                   "addrGen2":
                       // Выплнение команд генератора 2
                       REGION ADRES_GENERATOR 2     
                           CASE "GlobalDATA".REQ.CMD OF
                               "cmdSCUR":
                                   REGION SET_CURRENT
                                       //Установка тока генератора
                                       IF "GeneratorDATA_2".CMD_CP = FALSE THEN
                                           "GeneratorDATA_2".CP_Programm := "GlobalDATA".REQ.Value;
                                           "GeneratorDATA_2".CMD_CP := TRUE;
                                       END_IF;
                                       //Проверяем выполнение команды от генератора
                                       IF "GeneratorDATA_2".cmdDone = TRUE AND "GeneratorDATA_2".cmd_Nunmber = "FB_STATE_CURRENT_PROGRAMM" THEN
                                           "GlobalDATA".RESP.Value := "GeneratorDATA_2".CP_Programm;
                                           "GlobalDATA".RESP.Done := 1;
                                       ELSIF "GeneratorDATA_2".cmdError = TRUE THEN
                                           "GlobalDATA".RESP.Value := "GeneratorDATA_2".cmdState;
                                           "GlobalDATA".RESP.Done := 1;
                                       END_IF;
                                   END_REGION SET_CURRENT
                               "cmdSVLT":
                                   REGION SET_VOLTAGE
                                       //Устанавливаем напряжение генератора
                                       IF "GeneratorDATA_2".CMD_VP = FALSE THEN
                                           #TempReal := UINT_TO_REAL("GlobalDATA".REQ.Value);
                                           "GeneratorDATA_2".VP_Programm := #TempReal / 10.0;
                                           "GeneratorDATA_2".CMD_VP := TRUE;
                                       END_IF;
                                       //Проверяем выполнение команды от генератора
                                       IF "GeneratorDATA_2".cmdDone = TRUE AND "GeneratorDATA_2".cmd_Nunmber = "FB_STATE_VOLTAGE_PROGRAMM" THEN
                                           #TempReal := "GeneratorDATA_2".VP_Programm * 10.0;
                                           #TempUint := REAL_TO_UINT(#TempReal);
                                           "GlobalDATA".RESP.Value := #TempUint;
                                           "GlobalDATA".RESP.Done := 1;
                                       ELSIF "GeneratorDATA_2".cmdError = TRUE THEN
                                           "GlobalDATA".RESP.Value := "GeneratorDATA_2".cmdState;
                                           "GlobalDATA".RESP.Done := 1;
                                       END_IF;
                                   END_REGION SET_VOLTAGE
                               "cmdGCUR":
                                   REGION GET_CURRENT
                                       //Чтение тока генератора
                                       "GeneratorDATA_2".CMD_MON := TRUE;

                                       //Проверяем выполнение команды от генератора
                                       IF "GeneratorDATA_2".cmdDone = TRUE AND "GeneratorDATA_2".cmd_Nunmber = "FB_STATE_MONITOR" THEN
                                           "GlobalDATA".RESP.Value := "GeneratorDATA_2".CP_Monitor;
                                           "GlobalDATA".RESP.Done := 1;
                                       ELSIF "GeneratorDATA_2".cmdError = TRUE THEN
                                           "GlobalDATA".RESP.Value := "GeneratorDATA_2".cmdState;
                                           "GlobalDATA".RESP.Done := 1;
                                       END_IF;
                                   END_REGION GET_CURRENT
                               "cmdGVLT":
                                   REGION GET_VALUE
                                       //Чтение напряжения генератора
                                       "GeneratorDATA_2".CMD_MON := TRUE;

                                       //Проверяем выполнение команды от генератора
                                       IF "GeneratorDATA_2".cmdDone = TRUE AND "GeneratorDATA_2".cmd_Nunmber = "FB_STATE_MONITOR" THEN
                                           #TempReal := "GeneratorDATA_2".VP_Monitor * 10.0;
                                           #TempUint := REAL_TO_UINT(#TempReal);
                                           "GlobalDATA".RESP.Value := #TempUint;
                                           "GlobalDATA".RESP.Done := 1;
                                       ELSIF "GeneratorDATA_2".cmdError = TRUE THEN
                                           "GlobalDATA".RESP.Value := "GeneratorDATA_2".cmdState;
                                           "GlobalDATA".RESP.Done := 1;
                                       END_IF;
                                   END_REGION GET_VALUE
                               "cmdSRAY":
                                   REGION SET_XRAY
                                       //Включение X-RAY
                                       //Включение X-RAY если шторка находится в закрытом положении
                                       IF "GlobalDATA".Shutter2.setPOS1 OR "GlobalDATA".Shutter2.setPOS2 THEN
                                           IF "GlobalDATA".REQ.Value = 1 THEN
                                               "GlobalDATA".Generator2.CmdXRAY_ON := TRUE;
                                           ELSIF "GlobalDATA".REQ.Value = 0 THEN
                                               "GlobalDATA".Generator2.CmdXRAY_ON := FALSE;
                                           END_IF;

                                           //Проверяем статус генератора
                                           IF "GeneratorDATA_2".cmdDone = TRUE AND "GeneratorDATA_2".cmd_Nunmber = "FB_STATE_MONITOR" THEN
                                               IF ("GlobalDATA".REQ.Value = 1 AND "GlobalDATA".Generator2.XRAY_Status = TRUE) THEN
                                                   "GlobalDATA".RESP.Value := 1;
                                                   "GlobalDATA".RESP.Done := 1;
                                               END_IF;
                                               IF ("GlobalDATA".REQ.Value = 0 AND "GlobalDATA".Generator2.XRAY_Status = FALSE) THEN
                                                   "GlobalDATA".RESP.Value := 0;
                                                   "GlobalDATA".RESP.Done := 1;
                                               END_IF;
                                               IF "GeneratorDATA_2".cmdError = TRUE THEN
                                                   "GlobalDATA".RESP.Value := "GeneratorDATA_2".cmdState;
                                                   "GlobalDATA".RESP.Done := 1;
                                               END_IF;
                                           END_IF;
                                       ELSE
                                           "GlobalDATA".RESP.Value := "ERR_UNDEFINED_STATE";
                                           "GlobalDATA".RESP.Done := 1;
                                       END_IF;
                                   END_REGION SET_XRAY
                               "cmdGRAY":
                                   REGION GET_XRAY_STATUS
                                       //Проверяем статус генератора
                                       "GeneratorDATA_2".CMD_STAT := TRUE;
                                       IF "GeneratorDATA_2".cmdDone = TRUE AND "GeneratorDATA_2".cmd_Nunmber = "FB_STATE_HV_STATUS" THEN
                                           IF "GeneratorDATA_2".X_RAY_Status = TRUE THEN
                                               "GlobalDATA".RESP.Value := 1;
                                           ELSE
                                               "GlobalDATA".RESP.Value := 0;
                                           END_IF;
                                           "GlobalDATA".RESP.Done := 1;
                                       ELSIF "GeneratorDATA_2".cmdError = TRUE THEN
                                           "GlobalDATA".RESP.Value := "GeneratorDATA_2".cmdState;
                                           "GlobalDATA".REQ.CMD := 0;
                                       END_IF;
                                   END_REGION GET_XRAY_STATUS
                               "cmdSWAR":
                                   REGION SET_WARM
                                       //Установка режима прогрева генератора
                                       IF "GlobalDATA".Generator2.Ready = TRUE THEN
                                           "GlobalDATA".Generator2.cmdWarm := "GlobalDATA".REQ.Value;
                                           IF "GlobalDATA".Generator2.warmEN THEN
                                               "GlobalDATA".RESP.Done := 1;
                                               //Возвращаем код выполнения программы без ошибок
                                               "GlobalDATA".RESP.Value := "GlobalDATA".Generator2.cmdWarm;
                                           END_IF;
                                       ELSE
                                           //Если генератор был не готов, то выдаем ошибку
                                           "GlobalDATA".RESP.Done := 1;
                                           "GlobalDATA".RESP.Value := "ERR_UNDEFINED_STATE";
                                       END_IF;
                                   END_REGION SET_WARM
                               "cmdGWAR":
                                   REGION GET_WARM
                                       //Если генератор готов и идет прогрев, то возвращаем значение таблицы прогрева
                                       IF "GlobalDATA".Generator2.Ready = TRUE AND "GlobalDATA".Generator2.warmEN THEN
                                           //Возвращаем код выполнения программы без ошибок
                                           "GlobalDATA".RESP.Value := "GlobalDATA".Generator2.cmdWarm;
                                       ELSE
                                           //Если генератор был не готов или не выполняется прогрев, то выдаем ошибку
                                           "GlobalDATA".RESP.Value := "STATUS_NO_CALL";
                                       END_IF;
                                       "GlobalDATA".RESP.Done := 1;
                                   END_REGION GET_WARM
                               "cmdSCLR":
                                   REGION SET_CLEAR_FAULT
                                       //Сброс ошибок генератора
                                       "GeneratorDATA_2".CMD_CLR := TRUE;
                                       //Проверяем выполнение команды от генератора
                                       IF "GeneratorDATA_2".cmdDone = TRUE AND "GeneratorDATA_2".cmd_Nunmber = "FB_STATE_FAULT_CLEAR" THEN
                                           //Чтение ошибок генератора
                                           "GeneratorDATA_2".CMD_FLT := TRUE;
                                       END_IF;

                                       //Проверяем выполнение команды от генератора
                                       IF "GeneratorDATA_2".cmdDone = TRUE AND "GeneratorDATA_2".cmd_Nunmber = "FB_STATE_REPORT_FAULT" THEN
                                           "GlobalDATA".RESP.Value.%X0 := "GeneratorDATA_2".FLT[0];
                                           "GlobalDATA".RESP.Value.%X1 := "GeneratorDATA_2".FLT[1];
                                           "GlobalDATA".RESP.Value.%X2 := "GeneratorDATA_2".FLT[2];
                                           "GlobalDATA".RESP.Value.%X3 := "GeneratorDATA_2".FLT[3];
                                           "GlobalDATA".RESP.Value.%X4 := "GeneratorDATA_2".FLT[4];
                                           "GlobalDATA".RESP.Value.%X5 := "GeneratorDATA_2".FLT[5];
                                           "GlobalDATA".RESP.Value.%X6 := "GeneratorDATA_2".FLT[6];
                                           "GlobalDATA".RESP.Value.%X7 := "GeneratorDATA_2".FLT[7];
                                           "GlobalDATA".RESP.Value.%X8 := "GeneratorDATA_2".FLT[8];
                                           "GlobalDATA".RESP.Done := 1;
                                       ELSIF "GeneratorDATA_2".cmdError = TRUE THEN
                                           "GlobalDATA".RESP.Value := "GeneratorDATA_2".cmdState;
                                           "GlobalDATA".RESP.Done := 1;
                                       END_IF;
                                   END_REGION SET_CLEAR_FAULT
                               "cmdGFLT":
                                   REGION GET_FAULT
                                       //Чтение ошибок генератора
                                       "GeneratorDATA_2".CMD_FLT := TRUE;

                                       //Проверяем выполнение команды от генератора
                                       IF "GeneratorDATA_2".cmdDone = TRUE AND "GeneratorDATA_2".cmd_Nunmber = "FB_STATE_REPORT_FAULT" THEN
                                           "GlobalDATA".RESP.Value.%X0 := "GeneratorDATA_2".FLT[0];
                                           "GlobalDATA".RESP.Value.%X1 := "GeneratorDATA_2".FLT[1];
                                           "GlobalDATA".RESP.Value.%X2 := "GeneratorDATA_2".FLT[2];
                                           "GlobalDATA".RESP.Value.%X3 := "GeneratorDATA_2".FLT[3];
                                           "GlobalDATA".RESP.Value.%X4 := "GeneratorDATA_2".FLT[4];
                                           "GlobalDATA".RESP.Value.%X5 := "GeneratorDATA_2".FLT[5];
                                           "GlobalDATA".RESP.Value.%X6 := "GeneratorDATA_2".FLT[6];
                                           "GlobalDATA".RESP.Value.%X7 := "GeneratorDATA_2".FLT[7];
                                           "GlobalDATA".RESP.Value.%X8 := "GeneratorDATA_2".FLT[8];
                                           "GlobalDATA".RESP.Done := 1;
                                       ELSIF "GeneratorDATA_2".cmdError = TRUE THEN
                                           "GlobalDATA".RESP.Value := "GeneratorDATA_2".cmdState;
                                           "GlobalDATA".RESP.Done := 1;
                                       END_IF;
                                   END_REGION GET_FAULT
                               "cmdSRES":
                                   REGION SET_RESET
                                       //Выставляем признак сброса
                                       "GlobalDATA".cmdReset.Generator2 := TRUE;
                                       "GlobalDATA".RESP.Done := 1;
                                       "GlobalDATA".RESP.Value := "STATUS_SUBSEQUENT_CALL";
                                   END_REGION SET_RESET
                           END_CASE;
                       END_REGION ADRES_GENERATOR 2

                   "addrShutter1":
                       // Выплнение команд шторки 1
                       REGION ADRES_SHUTTER 1 
                           ;
                       END_REGION ADRES_SHUTTER 1

                   "addrShutter2":
                       // Выплнение команд шторки 2
                       REGION ADRES_SHUTTER 2    
                           ;
                       END_REGION ADRES_SHUTTER 2

                   "addrDoor":
                       // Выплнение команд двери
                       REGION ADRES_DOOR
                           CASE "GlobalDATA".REQ.CMD OF
                               "cmdSRES":
                                   REGION DriveDoorReset
                                       //Выставляем признак сброса
                                       "GlobalDATA".cmdReset.Door := TRUE;
                                       "GlobalDATA".RESP.Done := 1;
                                       "GlobalDATA".RESP.Value := "STATUS_SUBSEQUENT_CALL";
                                   END_REGION DriveDoorReset
                               ELSE  // Statement section ELSE
                                   ;
                           END_CASE;
                       END_REGION ADRES_DOOR

                   "addrDetector":
                       // Выплнение команд детекторов
                       REGION ADRES_DETECTOR    
                           CASE "GlobalDATA".REQ.CMD OF
                               "cmdSRES":
                                   REGION DetectorReset
                                       //Выставляем признак сброса
                                       "GlobalDATA".cmdReset.Detector := TRUE;
                                       "GlobalDATA".RESP.Done := 1;
                                       "GlobalDATA".RESP.Value := "STATUS_SUBSEQUENT_CALL";
                                   END_REGION DetectorReset
                               ELSE  // Statement section ELSE
                                   ;
                           END_CASE;
                       END_REGION ADRES_DETECTOR

                   "addrServoDrive1":
                       // Выполнение команд привода
                       REGION ADRES DRIVE1                      
                           CASE "GlobalDATA".REQ.CMD OF
                                   //КОманда на перемещение шторки
                               "cmdSPOS":
                                   //Даем команду на перемещение шторки
                                   IF "GlobalDATA".REQ.Value = 1 AND "TEL9_Drive1".driveStopped THEN
                                       "GlobalDATA".Shutter1.cmdPOS1 := TRUE;
                                   ELSIF "GlobalDATA".REQ.Value = 2 AND "TEL9_Drive1".driveStopped THEN
                                       "GlobalDATA".Shutter1.cmdPOS2 := TRUE;
                                   END_IF;

                                   //Проверяем положение шторки
                                   IF "GlobalDATA".REQ.Value = 1 AND "GlobalDATA".Shutter1.setPOS1 = TRUE AND "TEL9_Drive1".driveStopped = TRUE THEN
                                       "GlobalDATA".RESP.Done := 1;
                                       "GlobalDATA".RESP.Value := 1;
                                       "GlobalDATA".REQ.Value := 0;
                                   ELSIF "GlobalDATA".REQ.Value = 2 AND "GlobalDATA".Shutter1.setPOS2 = TRUE AND "TEL9_Drive1".driveStopped = TRUE THEN
                                       "GlobalDATA".RESP.Done := 1;
                                       "GlobalDATA".RESP.Value := 2;
                                       "GlobalDATA".REQ.Value := 0;
                                   END_IF;
                               "cmdSRES":
                                   REGION DriveReset
                                       //Выставляем признак сброса
                                       "GlobalDATA".cmdReset.Drive1 := TRUE;
                                       "GlobalDATA".RESP.Done := 1;
                                       "GlobalDATA".RESP.Value := "STATUS_SUBSEQUENT_CALL";
                                   END_REGION DriveReset   
                               ELSE  // Statement section ELSE
                                   ;
                           END_CASE;
                       END_REGION ADRES DRIVE1

                   "addrServoDrive2":
                       // Выполнение команд привода
                       REGION ADRES DRIVE2                      
                           CASE "GlobalDATA".REQ.CMD OF
                                   //КОманда на перемещение шторки
                               "cmdSPOS":
                                   //Даем команду на перемещение шторки
                                   IF "GlobalDATA".REQ.Value = 1 AND "TEL9_Drive2".driveStopped THEN
                                       "GlobalDATA".Shutter2.cmdPOS1 := TRUE;
                                   ELSIF "GlobalDATA".REQ.Value = 2 AND "TEL9_Drive2".driveStopped THEN
                                       "GlobalDATA".Shutter2.cmdPOS2 := TRUE;
                                   END_IF;

                                   //Проверяем положение шторки
                                   IF "GlobalDATA".REQ.Value = 1 AND "GlobalDATA".Shutter2.setPOS1 = TRUE AND "TEL9_Drive2".driveStopped = TRUE THEN
                                       "GlobalDATA".RESP.Done := 1;
                                       "GlobalDATA".RESP.Value := 1;
                                       "GlobalDATA".REQ.Value := 0;
                                   ELSIF "GlobalDATA".REQ.Value = 2 AND "GlobalDATA".Shutter2.setPOS2 = TRUE AND "TEL9_Drive2".driveStopped = TRUE THEN
                                       "GlobalDATA".RESP.Done := 1;
                                       "GlobalDATA".RESP.Value := 2;
                                       "GlobalDATA".REQ.Value := 0;
                                   END_IF;
                               "cmdSRES":
                                   REGION DriveReset
                                       //Выставляем признак сброса
                                       "GlobalDATA".cmdReset.Drive2 := TRUE;
                                       "GlobalDATA".RESP.Done := 1;
                                       "GlobalDATA".RESP.Value := "STATUS_SUBSEQUENT_CALL";
                                   END_REGION DriveReset   
                               ELSE  // Statement section ELSE
                                   ;
                           END_CASE;
                       END_REGION ADRES DRIVE2

                   ELSE  // Statement section ELSE
                       ;
               END_CASE;
           END_REGION ADDR_CMD_VALUE

   END_REGION STATE_RESPONCE
END_FUNCTION_BLOCK

FUNCTION "Val_to_Char" : Void   // FC7, SCL
{ S7_Optimized_Access := 'TRUE' }
VERSION : 0.1
   VAR_INPUT
      inValue : UInt;
   END_VAR
   VAR_OUTPUT
      charBUFF : Array[0..3] of Byte;
   END_VAR
   VAR_TEMP
      Countchar : UInt;
      StrValue : String;
      i : Int;
      tempBUFF : Array[0..3] of Byte;
      TEMP : UInt;
   END_VAR
BEGIN
   VAL_STRG(IN := #inValue,
            SIZE := 4,
            PREC := 0,
            FORMAT := 0,
            P := 1,
            OUT => #StrValue);

   #Countchar := 4;

   Strg_TO_Chars(Strg := #StrValue,
                 pChars := 0,
                 Cnt => #Countchar,
                 Chars := #tempBUFF);

   FOR #i := 0  TO 3 DO
      IF #tempBUFF[#i] = ' ' THEN // Statement section FOR
          #tempBUFF[#i] := '0';
       END_IF;
       #charBUFF[#i] := #tempBUFF[#i];
   END_FOR;
END_FUNCTION

// folder: DIO

FUNCTION "DI" : Void   // FC2, LAD
{ S7_Optimized_Access := 'TRUE' }
VERSION : 0.1
BEGIN

REGION Network 1: Чтение дискретных входов PLC и передача в глобальный блок данных
   // Первый байт дискретных входов
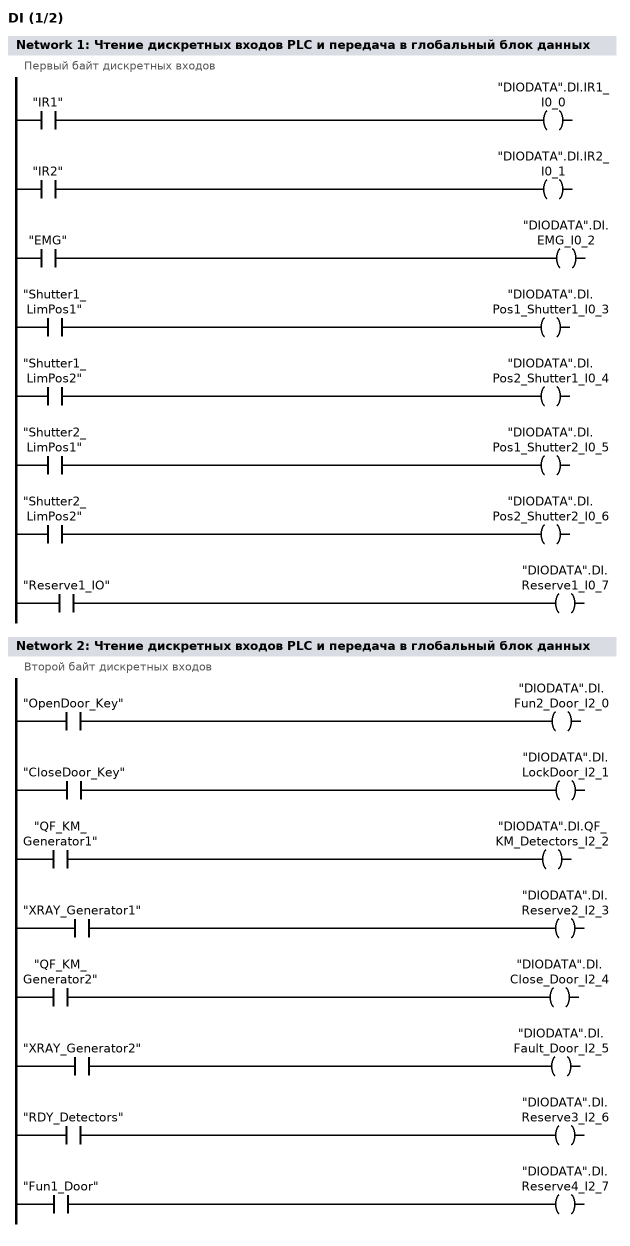
   RUNG wire#powerrail
      Contact( "IR1" )
      Coil( "DIODATA".DI.IR1_I0_0 )
   END_RUNG
   RUNG wire#powerrail
      Contact( "IR2" )
      Coil( "DIODATA".DI.IR2_I0_1 )
   END_RUNG
   RUNG wire#powerrail
      Contact( "EMG" )
      Coil( "DIODATA".DI.EMG_I0_2 )
   END_RUNG
   RUNG wire#powerrail
      Contact( "Shutter1_LimPos1" )
      Coil( "DIODATA".DI.Pos1_Shutter1_I0_3 )
   END_RUNG
   RUNG wire#powerrail
      Contact( "Shutter1_LimPos2" )
      Coil( "DIODATA".DI.Pos2_Shutter1_I0_4 )
   END_RUNG
   RUNG wire#powerrail
      Contact( "Shutter2_LimPos1" )
      Coil( "DIODATA".DI.Pos1_Shutter2_I0_5 )
   END_RUNG
   RUNG wire#powerrail
      Contact( "Shutter2_LimPos2" )
      Coil( "DIODATA".DI.Pos2_Shutter2_I0_6 )
   END_RUNG
   RUNG wire#powerrail
      Contact( "Reserve1_IO" )
      Coil( "DIODATA".DI.Reserve1_I0_7 )
   END_RUNG
   // the same network as SCL:
   "DIODATA".DI.IR1_I0_0 := "IR1";
   "DIODATA".DI.IR2_I0_1 := "IR2";
   "DIODATA".DI.EMG_I0_2 := "EMG";
   "DIODATA".DI.Pos1_Shutter1_I0_3 := "Shutter1_LimPos1";
   "DIODATA".DI.Pos2_Shutter1_I0_4 := "Shutter1_LimPos2";
   "DIODATA".DI.Pos1_Shutter2_I0_5 := "Shutter2_LimPos1";
   "DIODATA".DI.Pos2_Shutter2_I0_6 := "Shutter2_LimPos2";
   "DIODATA".DI.Reserve1_I0_7 := "Reserve1_IO";
END_REGION

REGION Network 2: Чтение дискретных входов PLC и передача в глобальный блок данных
   // Второй байт дискретных входов
   RUNG wire#powerrail
      Contact( "OpenDoor_Key" )
      Coil( "DIODATA".DI.Fun2_Door_I2_0 )
   END_RUNG
   RUNG wire#powerrail
      Contact( "CloseDoor_Key" )
      Coil( "DIODATA".DI.LockDoor_I2_1 )
   END_RUNG
   RUNG wire#powerrail
      Contact( "QF_KM_Generator1" )
      Coil( "DIODATA".DI.QF_KM_Detectors_I2_2 )
   END_RUNG
   RUNG wire#powerrail
      Contact( "XRAY_Generator1" )
      Coil( "DIODATA".DI.Reserve2_I2_3 )
   END_RUNG
   RUNG wire#powerrail
      Contact( "QF_KM_Generator2" )
      Coil( "DIODATA".DI.Close_Door_I2_4 )
   END_RUNG
   RUNG wire#powerrail
      Contact( "XRAY_Generator2" )
      Coil( "DIODATA".DI.Fault_Door_I2_5 )
   END_RUNG
   RUNG wire#powerrail
      Contact( "RDY_Detectors" )
      Coil( "DIODATA".DI.Reserve3_I2_6 )
   END_RUNG
   RUNG wire#powerrail
      Contact( "Fun1_Door" )
      Coil( "DIODATA".DI.Reserve4_I2_7 )
   END_RUNG
   // the same network as SCL:
   "DIODATA".DI.Fun2_Door_I2_0 := "OpenDoor_Key";
   "DIODATA".DI.LockDoor_I2_1 := "CloseDoor_Key";
   "DIODATA".DI.QF_KM_Detectors_I2_2 := "QF_KM_Generator1";
   "DIODATA".DI.Reserve2_I2_3 := "XRAY_Generator1";
   "DIODATA".DI.Close_Door_I2_4 := "QF_KM_Generator2";
   "DIODATA".DI.Fault_Door_I2_5 := "XRAY_Generator2";
   "DIODATA".DI.Reserve3_I2_6 := "RDY_Detectors";
   "DIODATA".DI.Reserve4_I2_7 := "Fun1_Door";
END_REGION

REGION Network 3: Чтение дискретных входов PLC и передача в глобальный блок данных
   // Третий
   //  байт дискретных входов
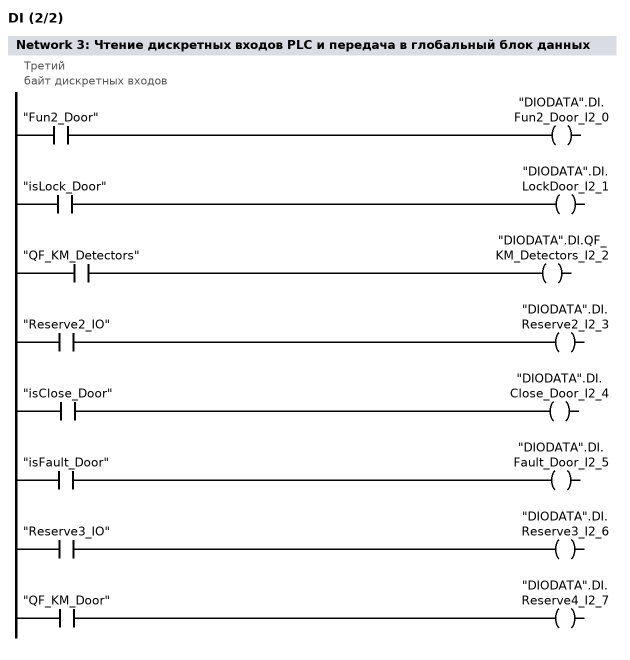
   RUNG wire#powerrail
      Contact( "Fun2_Door" )
      Coil( "DIODATA".DI.Fun2_Door_I2_0 )
   END_RUNG
   RUNG wire#powerrail
      Contact( "isLock_Door" )
      Coil( "DIODATA".DI.LockDoor_I2_1 )
   END_RUNG
   RUNG wire#powerrail
      Contact( "QF_KM_Detectors" )
      Coil( "DIODATA".DI.QF_KM_Detectors_I2_2 )
   END_RUNG
   RUNG wire#powerrail
      Contact( "Reserve2_IO" )
      Coil( "DIODATA".DI.Reserve2_I2_3 )
   END_RUNG
   RUNG wire#powerrail
      Contact( "isClose_Door" )
      Coil( "DIODATA".DI.Close_Door_I2_4 )
   END_RUNG
   RUNG wire#powerrail
      Contact( "isFault_Door" )
      Coil( "DIODATA".DI.Fault_Door_I2_5 )
   END_RUNG
   RUNG wire#powerrail
      Contact( "Reserve3_IO" )
      Coil( "DIODATA".DI.Reserve3_I2_6 )
   END_RUNG
   RUNG wire#powerrail
      Contact( "QF_KM_Door" )
      Coil( "DIODATA".DI.Reserve4_I2_7 )
   END_RUNG
   // the same network as SCL:
   "DIODATA".DI.Fun2_Door_I2_0 := "Fun2_Door";
   "DIODATA".DI.LockDoor_I2_1 := "isLock_Door";
   "DIODATA".DI.QF_KM_Detectors_I2_2 := "QF_KM_Detectors";
   "DIODATA".DI.Reserve2_I2_3 := "Reserve2_IO";
   "DIODATA".DI.Close_Door_I2_4 := "isClose_Door";
   "DIODATA".DI.Fault_Door_I2_5 := "isFault_Door";
   "DIODATA".DI.Reserve3_I2_6 := "Reserve3_IO";
   "DIODATA".DI.Reserve4_I2_7 := "QF_KM_Door";
END_REGION
END_FUNCTION

FUNCTION "DO" : Void   // FC6, LAD
{ S7_Optimized_Access := 'TRUE' }
VERSION : 0.1
BEGIN

REGION Network 1: Установка дискретных выходов PLC из глобального блока данных
   // Установка первого байта цифровых выходов
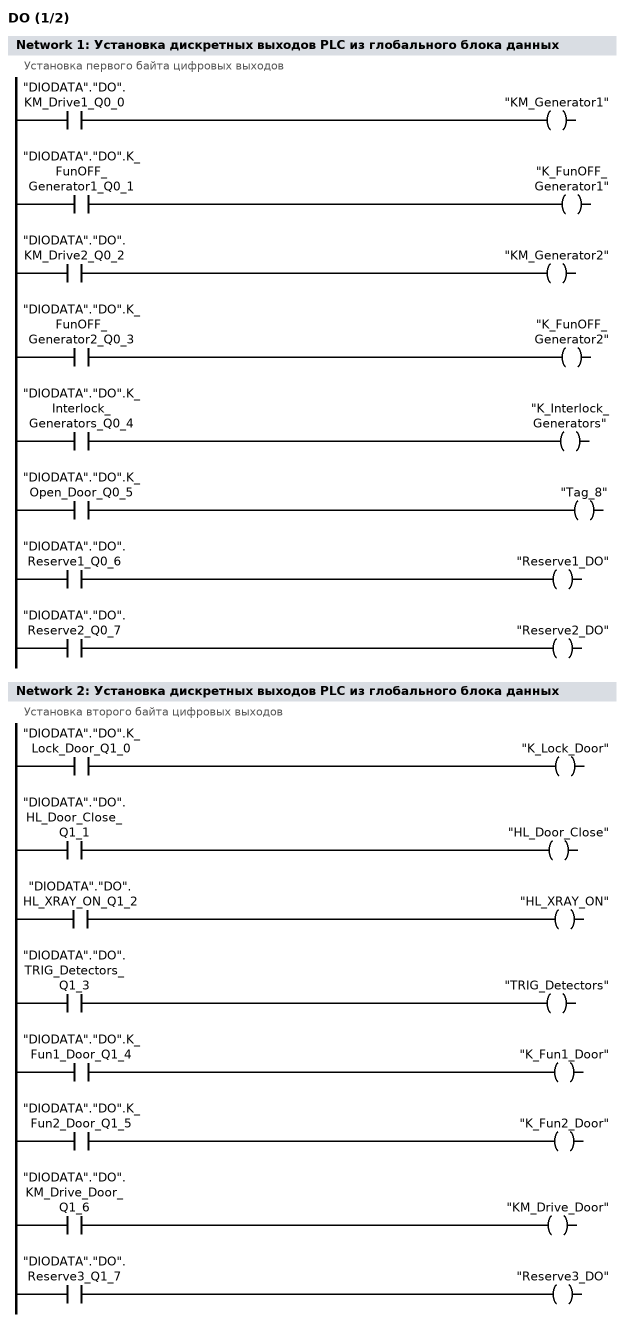
   RUNG wire#powerrail
      Contact( "DIODATA"."DO".KM_Drive1_Q0_0 )
      Coil( "KM_Generator1" )
   END_RUNG
   RUNG wire#powerrail
      Contact( "DIODATA"."DO".K_FunOFF_Generator1_Q0_1 )
      Coil( "K_FunOFF_Generator1" )
   END_RUNG
   RUNG wire#powerrail
      Contact( "DIODATA"."DO".KM_Drive2_Q0_2 )
      Coil( "KM_Generator2" )
   END_RUNG
   RUNG wire#powerrail
      Contact( "DIODATA"."DO".K_FunOFF_Generator2_Q0_3 )
      Coil( "K_FunOFF_Generator2" )
   END_RUNG
   RUNG wire#powerrail
      Contact( "DIODATA"."DO".K_Interlock_Generators_Q0_4 )
      Coil( "K_Interlock_Generators" )
   END_RUNG
   RUNG wire#powerrail
      Contact( "DIODATA"."DO".K_Open_Door_Q0_5 )
      Coil( "Tag_8" )
   END_RUNG
   RUNG wire#powerrail
      Contact( "DIODATA"."DO".Reserve1_Q0_6 )
      Coil( "Reserve1_DO" )
   END_RUNG
   RUNG wire#powerrail
      Contact( "DIODATA"."DO".Reserve2_Q0_7 )
      Coil( "Reserve2_DO" )
   END_RUNG
   // the same network as SCL:
   "KM_Generator1" := "DIODATA"."DO".KM_Drive1_Q0_0;
   "K_FunOFF_Generator1" := "DIODATA"."DO".K_FunOFF_Generator1_Q0_1;
   "KM_Generator2" := "DIODATA"."DO".KM_Drive2_Q0_2;
   "K_FunOFF_Generator2" := "DIODATA"."DO".K_FunOFF_Generator2_Q0_3;
   "K_Interlock_Generators" := "DIODATA"."DO".K_Interlock_Generators_Q0_4;
   "Tag_8" := "DIODATA"."DO".K_Open_Door_Q0_5;
   "Reserve1_DO" := "DIODATA"."DO".Reserve1_Q0_6;
   "Reserve2_DO" := "DIODATA"."DO".Reserve2_Q0_7;
END_REGION

REGION Network 2: Установка дискретных выходов PLC из глобального блока данных
   // Установка второго байта цифровых выходов
   RUNG wire#powerrail
      Contact( "DIODATA"."DO".K_Lock_Door_Q1_0 )
      Coil( "K_Lock_Door" )
   END_RUNG
   RUNG wire#powerrail
      Contact( "DIODATA"."DO".HL_Door_Close_Q1_1 )
      Coil( "HL_Door_Close" )
   END_RUNG
   RUNG wire#powerrail
      Contact( "DIODATA"."DO".HL_XRAY_ON_Q1_2 )
      Coil( "HL_XRAY_ON" )
   END_RUNG
   RUNG wire#powerrail
      Contact( "DIODATA"."DO".TRIG_Detectors_Q1_3 )
      Coil( "TRIG_Detectors" )
   END_RUNG
   RUNG wire#powerrail
      Contact( "DIODATA"."DO".K_Fun1_Door_Q1_4 )
      Coil( "K_Fun1_Door" )
   END_RUNG
   RUNG wire#powerrail
      Contact( "DIODATA"."DO".K_Fun2_Door_Q1_5 )
      Coil( "K_Fun2_Door" )
   END_RUNG
   RUNG wire#powerrail
      Contact( "DIODATA"."DO".KM_Drive_Door_Q1_6 )
      Coil( "KM_Drive_Door" )
   END_RUNG
   RUNG wire#powerrail
      Contact( "DIODATA"."DO".Reserve3_Q1_7 )
      Coil( "Reserve3_DO" )
   END_RUNG
   // the same network as SCL:
   "K_Lock_Door" := "DIODATA"."DO".K_Lock_Door_Q1_0;
   "HL_Door_Close" := "DIODATA"."DO".HL_Door_Close_Q1_1;
   "HL_XRAY_ON" := "DIODATA"."DO".HL_XRAY_ON_Q1_2;
   "TRIG_Detectors" := "DIODATA"."DO".TRIG_Detectors_Q1_3;
   "K_Fun1_Door" := "DIODATA"."DO".K_Fun1_Door_Q1_4;
   "K_Fun2_Door" := "DIODATA"."DO".K_Fun2_Door_Q1_5;
   "KM_Drive_Door" := "DIODATA"."DO".KM_Drive_Door_Q1_6;
   "Reserve3_DO" := "DIODATA"."DO".Reserve3_Q1_7;
END_REGION

REGION Network 3: Установка дискретных выходов PLC из глобального блока данных
   // Установка третьего байта цифровых выходов
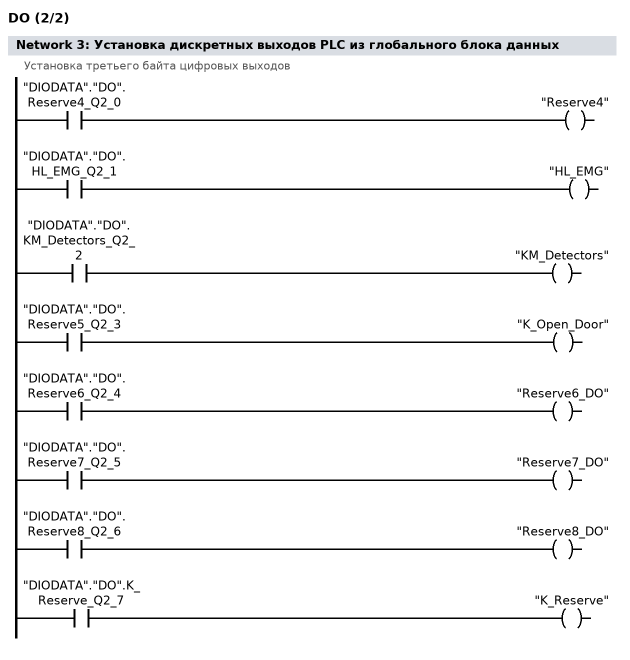
   RUNG wire#powerrail
      Contact( "DIODATA"."DO".Reserve4_Q2_0 )
      Coil( "Reserve4" )
   END_RUNG
   RUNG wire#powerrail
      Contact( "DIODATA"."DO".HL_EMG_Q2_1 )
      Coil( "HL_EMG" )
   END_RUNG
   RUNG wire#powerrail
      Contact( "DIODATA"."DO".KM_Detectors_Q2_2 )
      Coil( "KM_Detectors" )
   END_RUNG
   RUNG wire#powerrail
      Contact( "DIODATA"."DO".Reserve5_Q2_3 )
      Coil( "K_Open_Door" )
   END_RUNG
   RUNG wire#powerrail
      Contact( "DIODATA"."DO".Reserve6_Q2_4 )
      Coil( "Reserve6_DO" )
   END_RUNG
   RUNG wire#powerrail
      Contact( "DIODATA"."DO".Reserve7_Q2_5 )
      Coil( "Reserve7_DO" )
   END_RUNG
   RUNG wire#powerrail
      Contact( "DIODATA"."DO".Reserve8_Q2_6 )
      Coil( "Reserve8_DO" )
   END_RUNG
   RUNG wire#powerrail
      Contact( "DIODATA"."DO".K_Reserve_Q2_7 )
      Coil( "K_Reserve" )
   END_RUNG
   // the same network as SCL:
   "Reserve4" := "DIODATA"."DO".Reserve4_Q2_0;
   "HL_EMG" := "DIODATA"."DO".HL_EMG_Q2_1;
   "KM_Detectors" := "DIODATA"."DO".KM_Detectors_Q2_2;
   "K_Open_Door" := "DIODATA"."DO".Reserve5_Q2_3;
   "Reserve6_DO" := "DIODATA"."DO".Reserve6_Q2_4;
   "Reserve7_DO" := "DIODATA"."DO".Reserve7_Q2_5;
   "Reserve8_DO" := "DIODATA"."DO".Reserve8_Q2_6;
   "K_Reserve" := "DIODATA"."DO".K_Reserve_Q2_7;
END_REGION
END_FUNCTION

// folder: Drive

FUNCTION_BLOCK "DrivesStage"   // FB2, LAD
{ S7_Optimized_Access := 'TRUE' }
VERSION : 0.1
   VAR_INPUT
      Drive1 : Bool;   // drive 1 manage
      Drive2 : Bool;   // drive 1 manage
      Resset : Bool;   // Resset Block
      Mode : Bool;   // 0-MDI, 1-JOG
      "ON/OFF1" : Bool;   // OFF1
      JOG1 : Bool;   // JOG+
      JOG2 : Bool;   // JOG-
      cmdPOS1 : Bool;   // position to point 1
      cmdPOS2 : Bool;   // position to point 2
      Velocity : DInt;   // Velocity in MDI
      accelerationOverride : Real;   // accelerationOverride %
      decelerationOverride : Real;   // decelerationOverride %
      POS1_X : DInt;   // coordinate of point 1
      POS2_X : DInt;   // coordinate of point 2
      CmdPOS : Bool;   // CMD to traversing task
      HardWare_IO : Hw_Io;   // Hardware identifer of the drive axis
   END_VAR
   VAR_OUTPUT
      State_OFF1 : Bool;   // State OFF1
      Drive_STOP : Bool;   // State Drive Stop
      setPOS1 : Bool;   // in position 1
      setPOS2 : Bool;   // in position 2
      actualPosition : DInt;   // Current position
      Fault_Active : Bool;   // Fault Active
   END_VAR
   VAR_IN_OUT
      DATA : "typeTEL9";
   END_VAR
   VAR
      sSetPOS : Bool;
      sOFF1 : Bool;
      sOFF2 : Bool;
      sOFF3 : Bool;
      Front1 : Bool;
      Front2 : Bool;
      Front3 : Bool;
      Task : UInt;
      neg1 : Bool;
   END_VAR
   VAR_TEMP
      In_pos1 : Bool;
      In_pos2 : Bool;
   END_VAR
   VAR_TEMP   // added for the SCL form of the ladder/FBD networks
      _w1 : Bool;
      _w2 : Bool;
   END_VAR
BEGIN

REGION Network 1: Включение OFF1. Если возникает ошибка привода, то снимаем OFF1, сбрасываем ошибку и опять ввзводим OFF1
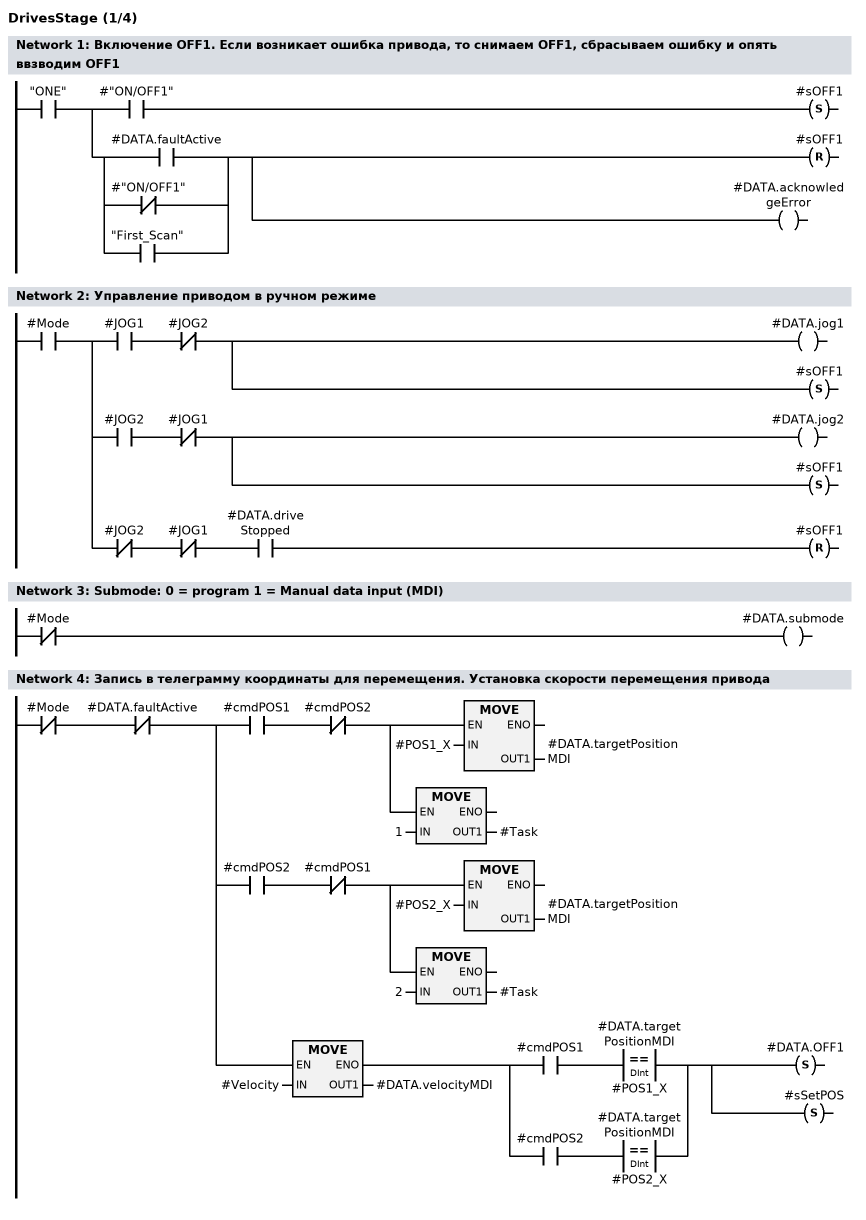
   RUNG wire#powerrail
      Contact( "ONE" )
      wire#w1
      Contact( #"ON/OFF1" )
      S_Coil( #sOFF1 )
   END_RUNG
   RUNG wire#w1
      Contact( #DATA.faultActive )
      wire#w2
      R_Coil( #sOFF1 )
   END_RUNG
   RUNG wire#w1
      I_Contact( #"ON/OFF1" )
   END_RUNG wire#w2
   RUNG wire#w1
      Contact( "First_Scan" )
   END_RUNG wire#w2
   RUNG wire#w2
      Coil( #DATA.acknowledgeError )
   END_RUNG
   // the same network as SCL:
   IF "ONE" AND #"ON/OFF1" THEN #sOFF1 := TRUE; END_IF;
   #_w1 := "ONE" AND (#DATA.faultActive OR NOT #"ON/OFF1" OR "First_Scan");
   IF #_w1 THEN #sOFF1 := FALSE; END_IF;
   #DATA.acknowledgeError := #_w1;
END_REGION

REGION Network 2: Управление приводом в ручном режиме
   RUNG wire#powerrail
      Contact( #Mode )
      wire#w1
      Contact( #JOG1 )
      I_Contact( #JOG2 )
      wire#w2
      Coil( #DATA.jog1 )
   END_RUNG
   RUNG wire#w2
      S_Coil( #sOFF1 )
   END_RUNG
   RUNG wire#w1
      Contact( #JOG2 )
      I_Contact( #JOG1 )
      wire#w3
      Coil( #DATA.jog2 )
   END_RUNG
   RUNG wire#w3
      S_Coil( #sOFF1 )
   END_RUNG
   RUNG wire#w1
      I_Contact( #JOG2 )
      I_Contact( #JOG1 )
      Contact( #DATA.driveStopped )
      R_Coil( #sOFF1 )
   END_RUNG
   // the same network as SCL:
   #DATA.jog1 := #Mode AND #JOG1 AND NOT #JOG2;
   IF #DATA.jog1 THEN #sOFF1 := TRUE; END_IF;
   #DATA.jog2 := #Mode AND #JOG2 AND NOT #JOG1;
   IF #DATA.jog2 THEN #sOFF1 := TRUE; END_IF;
   IF #Mode AND NOT #JOG2 AND NOT #JOG1 AND #DATA.driveStopped THEN #sOFF1 := FALSE; END_IF;
END_REGION

REGION Network 3: Submode: 0 = program 1 = Manual data input (MDI)
   RUNG wire#powerrail
      I_Contact( #Mode )
      Coil( #DATA.submode )
   END_RUNG
   // the same network as SCL:
   #DATA.submode := NOT #Mode;
END_REGION

REGION Network 4: Запись в телеграмму координаты для перемещения. Установка скорости перемещения привода
   RUNG wire#powerrail
      I_Contact( #Mode )
      I_Contact( #DATA.faultActive )
      wire#w1
      Contact( #cmdPOS1 )
      I_Contact( #cmdPOS2 )
      wire#w2
      Move(in := #POS1_X, out1 => #DATA.targetPositionMDI)
   END_RUNG
   RUNG wire#w2
      Move(in := 1, out1 => #Task)
   END_RUNG
   RUNG wire#w1
      Contact( #cmdPOS2 )
      I_Contact( #cmdPOS1 )
      wire#w3
      Move(in := #POS2_X, out1 => #DATA.targetPositionMDI)
   END_RUNG
   RUNG wire#w3
      Move(in := 2, out1 => #Task)
   END_RUNG
   RUNG wire#w1
      Move(in := #Velocity, out1 => #DATA.velocityMDI)
      wire#w4
      Contact( #cmdPOS1 )
      { S7_Templates := "SrcType := DInt" } EQ_Contact(in1 := #DATA.targetPositionMDI, in2 := #POS1_X)
      wire#w5
      S_Coil( #DATA.OFF1 )
   END_RUNG
   RUNG wire#w4
      Contact( #cmdPOS2 )
      { S7_Templates := "SrcType := DInt" } EQ_Contact(in1 := #DATA.targetPositionMDI, in2 := #POS2_X)
   END_RUNG wire#w5
   RUNG wire#w5
      S_Coil( #sSetPOS )
   END_RUNG
   // the same network as SCL:
   #_w1 := NOT #Mode AND NOT #DATA.faultActive;
   IF #_w1 AND #cmdPOS1 AND NOT #cmdPOS2 THEN
       #DATA.targetPositionMDI := #POS1_X;
       #Task := 1;
   END_IF;
   IF #_w1 AND #cmdPOS2 AND NOT #cmdPOS1 THEN
       #DATA.targetPositionMDI := #POS2_X;
       #Task := 2;
   END_IF;
   IF #_w1 THEN #DATA.velocityMDI := #Velocity; END_IF;
   IF #_w1 AND ((#cmdPOS1 AND (#DATA.targetPositionMDI = #POS1_X)) OR (#cmdPOS2 AND (#DATA.targetPositionMDI = #POS2_X))) THEN
       #DATA.OFF1 := TRUE;
       #sSetPOS := TRUE;
   END_IF;
END_REGION

REGION Network 5: Activate traversing task
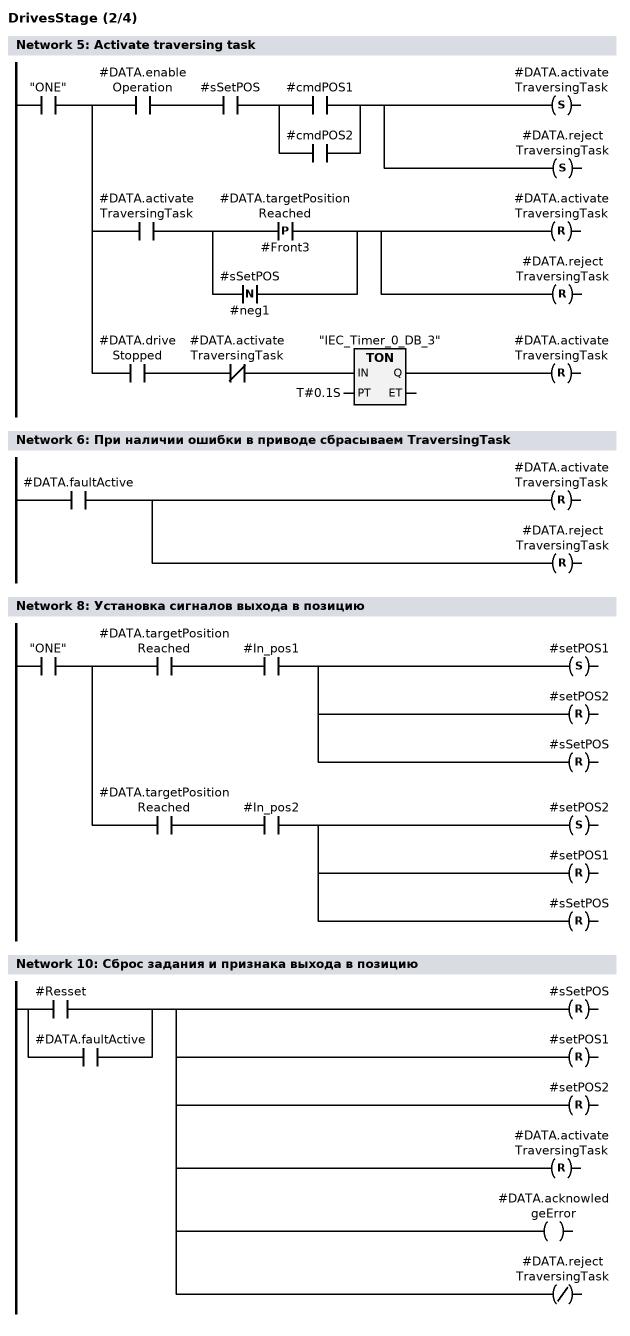
   IF "ONE" AND #DATA.enableOperation AND #sSetPOS AND (#cmdPOS1 OR #cmdPOS2) THEN
       #DATA.activateTraversingTask := TRUE;
       #DATA.rejectTraversingTask := TRUE;
   END_IF;
   #_w1 := "ONE" AND #DATA.activateTraversingTask AND #DATA.targetPositionReached AND NOT #Front3;   // rising edge of #DATA.targetPositionReached
   #Front3 := #DATA.targetPositionReached;
   #_w2 := "ONE" AND #DATA.activateTraversingTask AND NOT #sSetPOS AND #neg1;   // falling edge of #sSetPOS
   #neg1 := #sSetPOS;
   IF #_w1 OR #_w2 THEN
       #DATA.activateTraversingTask := FALSE;
       #DATA.rejectTraversingTask := FALSE;
   END_IF;
   "IEC_Timer_0_DB_3".TON(IN := "ONE" AND #DATA.driveStopped AND NOT #DATA.activateTraversingTask, PT := T#0.1S);
   IF "IEC_Timer_0_DB_3".Q THEN #DATA.activateTraversingTask := FALSE; END_IF;
END_REGION

REGION Network 6: При наличии ошибки в приводе сбрасываем TraversingTask
   RUNG wire#powerrail
      Contact( #DATA.faultActive )
      wire#w1
      R_Coil( #DATA.activateTraversingTask )
   END_RUNG
   RUNG wire#w1
      R_Coil( #DATA.rejectTraversingTask )
   END_RUNG
   // the same network as SCL:
   IF #DATA.faultActive THEN
       #DATA.activateTraversingTask := FALSE;
       #DATA.rejectTraversingTask := FALSE;
   END_IF;
END_REGION

REGION Network 7 (SCL)
   IF ABS(#DATA.actualPosition-#POS1_X)<40 THEN
       #In_pos1 := TRUE;
   ELSE
       #In_pos1 := FALSE;
   END_IF;
   IF  ABS(#DATA.actualPosition - #POS2_X) < 40 THEN
       #In_pos2 := TRUE;
   ELSE
       #In_pos2 := FALSE;
   END_IF;
END_REGION

REGION Network 8: Установка сигналов выхода в позицию
   RUNG wire#powerrail
      Contact( "ONE" )
      wire#w1
      Contact( #DATA.targetPositionReached )
      Contact( #In_pos1 )
      wire#w2
      S_Coil( #setPOS1 )
   END_RUNG
   RUNG wire#w2
      R_Coil( #setPOS2 )
   END_RUNG
   RUNG wire#w2
      R_Coil( #sSetPOS )
   END_RUNG
   RUNG wire#w1
      Contact( #DATA.targetPositionReached )
      Contact( #In_pos2 )
      wire#w3
      S_Coil( #setPOS2 )
   END_RUNG
   RUNG wire#w3
      R_Coil( #setPOS1 )
   END_RUNG
   RUNG wire#w3
      R_Coil( #sSetPOS )
   END_RUNG
   // the same network as SCL:
   IF "ONE" AND #DATA.targetPositionReached AND #In_pos1 THEN
       #setPOS1 := TRUE;
       #setPOS2 := FALSE;
       #sSetPOS := FALSE;
   END_IF;
   IF "ONE" AND #DATA.targetPositionReached AND #In_pos2 THEN
       #setPOS2 := TRUE;
       #setPOS1 := FALSE;
       #sSetPOS := FALSE;
   END_IF;
END_REGION

REGION Network 9 (SCL)
   #DATA.positioningModeMDI := 1;
   #DATA.intermediateStop := TRUE;
   #Task := 0;
END_REGION

REGION Network 10: Сброс задания и признака выхода в позицию
   RUNG wire#powerrail
      Contact( #Resset )
      wire#w1
      R_Coil( #sSetPOS )
   END_RUNG
   RUNG wire#powerrail
      Contact( #DATA.faultActive )
   END_RUNG wire#w1
   RUNG wire#w1
      R_Coil( #setPOS1 )
   END_RUNG
   RUNG wire#w1
      R_Coil( #setPOS2 )
   END_RUNG
   RUNG wire#w1
      R_Coil( #DATA.activateTraversingTask )
   END_RUNG
   RUNG wire#w1
      Coil( #DATA.acknowledgeError )
   END_RUNG
   RUNG wire#w1
      I_Coil( #DATA.rejectTraversingTask )
   END_RUNG
   // the same network as SCL:
   #_w1 := #Resset OR #DATA.faultActive;
   IF #_w1 THEN
       #sSetPOS := FALSE;
       #setPOS1 := FALSE;
       #setPOS2 := FALSE;
       #DATA.activateTraversingTask := FALSE;
   END_IF;
   #DATA.acknowledgeError := #_w1;
   #DATA.rejectTraversingTask := NOT #_w1;
END_REGION

REGION Network 11: Формирование телеграммы для привода
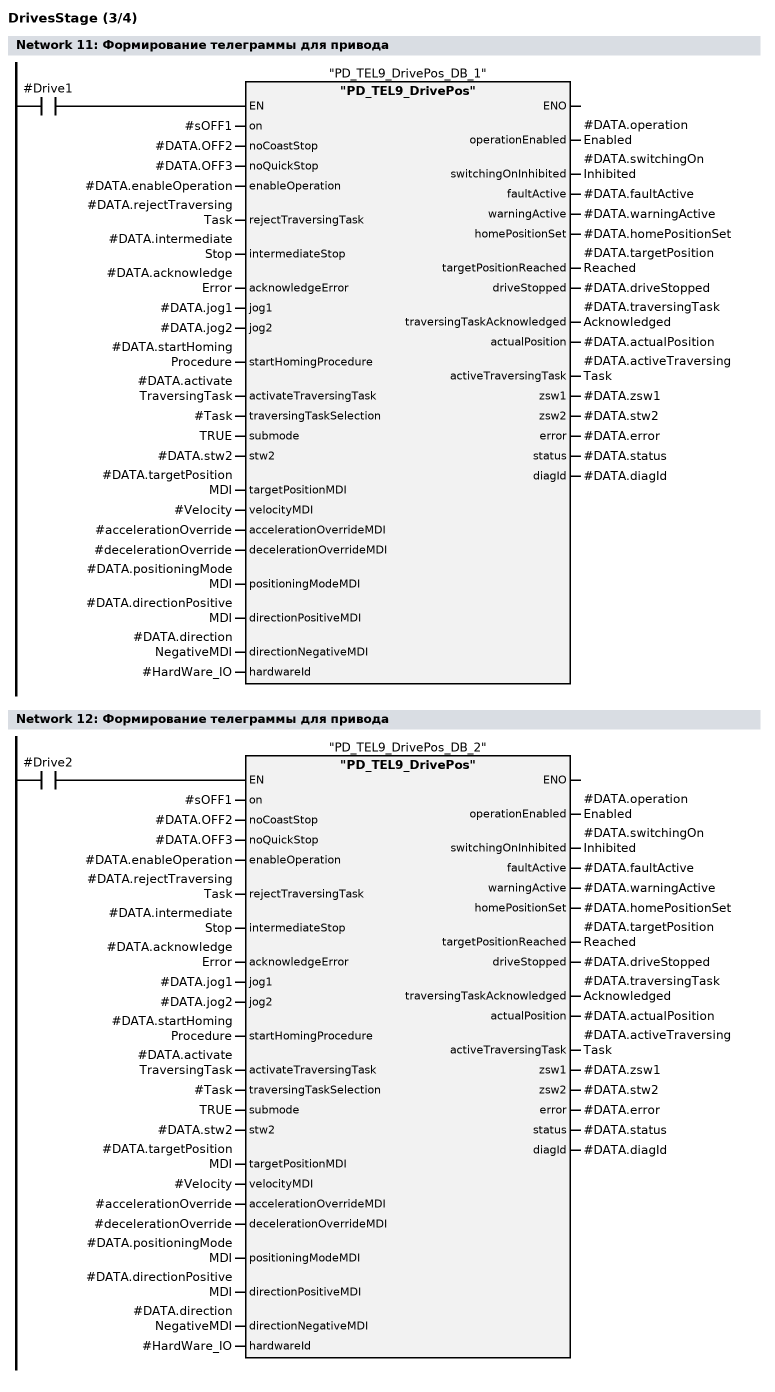
   RUNG wire#powerrail
      Contact( #Drive1 )
      "PD_TEL9_DrivePos_DB_1"(on := #sOFF1, noCoastStop := #DATA.OFF2, noQuickStop := #DATA.OFF3, enableOperation := #DATA.enableOperation, rejectTraversingTask := #DATA.rejectTraversingTask, intermediateStop := #DATA.intermediateStop, acknowledgeError := #DATA.acknowledgeError, jog1 := #DATA.jog1, jog2 := #DATA.jog2, startHomingProcedure := #DATA.startHomingProcedure, activateTraversingTask := #DATA.activateTraversingTask, traversingTaskSelection := #Task, submode := TRUE, stw2 := #DATA.stw2, targetPositionMDI := #DATA.targetPositionMDI, velocityMDI := #Velocity, accelerationOverrideMDI := #accelerationOverride, decelerationOverrideMDI := #decelerationOverride, positioningModeMDI := #DATA.positioningModeMDI, directionPositiveMDI := #DATA.directionPositiveMDI, directionNegativeMDI := #DATA.directionNegativeMDI, hardwareId := #HardWare_IO, operationEnabled => #DATA.operationEnabled, switchingOnInhibited => #DATA.switchingOnInhibited, faultActive => #DATA.faultActive, warningActive => #DATA.warningActive, homePositionSet => #DATA.homePositionSet, targetPositionReached => #DATA.targetPositionReached, driveStopped => #DATA.driveStopped, traversingTaskAcknowledged => #DATA.traversingTaskAcknowledged, actualPosition => #DATA.actualPosition, activeTraversingTask => #DATA.activeTraversingTask, zsw1 => #DATA.zsw1, zsw2 => #DATA.stw2, error => #DATA.error, status => #DATA.status, diagId => #DATA.diagId)
   END_RUNG
   // the same network as SCL:
   IF #Drive1 THEN
       "PD_TEL9_DrivePos_DB_1"(on := #sOFF1,   // "PD_TEL9_DrivePos"
                               noCoastStop := #DATA.OFF2,
                               noQuickStop := #DATA.OFF3,
                               enableOperation := #DATA.enableOperation,
                               rejectTraversingTask := #DATA.rejectTraversingTask,
                               intermediateStop := #DATA.intermediateStop,
                               acknowledgeError := #DATA.acknowledgeError,
                               jog1 := #DATA.jog1,
                               jog2 := #DATA.jog2,
                               startHomingProcedure := #DATA.startHomingProcedure,
                               activateTraversingTask := #DATA.activateTraversingTask,
                               traversingTaskSelection := #Task,
                               submode := TRUE,
                               stw2 := #DATA.stw2,
                               targetPositionMDI := #DATA.targetPositionMDI,
                               velocityMDI := #Velocity,
                               accelerationOverrideMDI := #accelerationOverride,
                               decelerationOverrideMDI := #decelerationOverride,
                               positioningModeMDI := #DATA.positioningModeMDI,
                               directionPositiveMDI := #DATA.directionPositiveMDI,
                               directionNegativeMDI := #DATA.directionNegativeMDI,
                               hardwareId := #HardWare_IO,
                               operationEnabled => #DATA.operationEnabled,
                               switchingOnInhibited => #DATA.switchingOnInhibited,
                               faultActive => #DATA.faultActive,
                               warningActive => #DATA.warningActive,
                               homePositionSet => #DATA.homePositionSet,
                               targetPositionReached => #DATA.targetPositionReached,
                               driveStopped => #DATA.driveStopped,
                               traversingTaskAcknowledged => #DATA.traversingTaskAcknowledged,
                               actualPosition => #DATA.actualPosition,
                               activeTraversingTask => #DATA.activeTraversingTask,
                               zsw1 => #DATA.zsw1,
                               zsw2 => #DATA.stw2,
                               error => #DATA.error,
                               status => #DATA.status,
                               diagId => #DATA.diagId);
   END_IF;
END_REGION

REGION Network 12: Формирование телеграммы для привода
   RUNG wire#powerrail
      Contact( #Drive2 )
      "PD_TEL9_DrivePos_DB_2"(on := #sOFF1, noCoastStop := #DATA.OFF2, noQuickStop := #DATA.OFF3, enableOperation := #DATA.enableOperation, rejectTraversingTask := #DATA.rejectTraversingTask, intermediateStop := #DATA.intermediateStop, acknowledgeError := #DATA.acknowledgeError, jog1 := #DATA.jog1, jog2 := #DATA.jog2, startHomingProcedure := #DATA.startHomingProcedure, activateTraversingTask := #DATA.activateTraversingTask, traversingTaskSelection := #Task, submode := TRUE, stw2 := #DATA.stw2, targetPositionMDI := #DATA.targetPositionMDI, velocityMDI := #Velocity, accelerationOverrideMDI := #accelerationOverride, decelerationOverrideMDI := #decelerationOverride, positioningModeMDI := #DATA.positioningModeMDI, directionPositiveMDI := #DATA.directionPositiveMDI, directionNegativeMDI := #DATA.directionNegativeMDI, hardwareId := #HardWare_IO, operationEnabled => #DATA.operationEnabled, switchingOnInhibited => #DATA.switchingOnInhibited, faultActive => #DATA.faultActive, warningActive => #DATA.warningActive, homePositionSet => #DATA.homePositionSet, targetPositionReached => #DATA.targetPositionReached, driveStopped => #DATA.driveStopped, traversingTaskAcknowledged => #DATA.traversingTaskAcknowledged, actualPosition => #DATA.actualPosition, activeTraversingTask => #DATA.activeTraversingTask, zsw1 => #DATA.zsw1, zsw2 => #DATA.stw2, error => #DATA.error, status => #DATA.status, diagId => #DATA.diagId)
   END_RUNG
   // the same network as SCL:
   IF #Drive2 THEN
       "PD_TEL9_DrivePos_DB_2"(on := #sOFF1,   // "PD_TEL9_DrivePos"
                               noCoastStop := #DATA.OFF2,
                               noQuickStop := #DATA.OFF3,
                               enableOperation := #DATA.enableOperation,
                               rejectTraversingTask := #DATA.rejectTraversingTask,
                               intermediateStop := #DATA.intermediateStop,
                               acknowledgeError := #DATA.acknowledgeError,
                               jog1 := #DATA.jog1,
                               jog2 := #DATA.jog2,
                               startHomingProcedure := #DATA.startHomingProcedure,
                               activateTraversingTask := #DATA.activateTraversingTask,
                               traversingTaskSelection := #Task,
                               submode := TRUE,
                               stw2 := #DATA.stw2,
                               targetPositionMDI := #DATA.targetPositionMDI,
                               velocityMDI := #Velocity,
                               accelerationOverrideMDI := #accelerationOverride,
                               decelerationOverrideMDI := #decelerationOverride,
                               positioningModeMDI := #DATA.positioningModeMDI,
                               directionPositiveMDI := #DATA.directionPositiveMDI,
                               directionNegativeMDI := #DATA.directionNegativeMDI,
                               hardwareId := #HardWare_IO,
                               operationEnabled => #DATA.operationEnabled,
                               switchingOnInhibited => #DATA.switchingOnInhibited,
                               faultActive => #DATA.faultActive,
                               warningActive => #DATA.warningActive,
                               homePositionSet => #DATA.homePositionSet,
                               targetPositionReached => #DATA.targetPositionReached,
                               driveStopped => #DATA.driveStopped,
                               traversingTaskAcknowledged => #DATA.traversingTaskAcknowledged,
                               actualPosition => #DATA.actualPosition,
                               activeTraversingTask => #DATA.activeTraversingTask,
                               zsw1 => #DATA.zsw1,
                               zsw2 => #DATA.stw2,
                               error => #DATA.error,
                               status => #DATA.status,
                               diagId => #DATA.diagId);
   END_IF;
END_REGION

REGION Network 13: Формирование выходных переменных
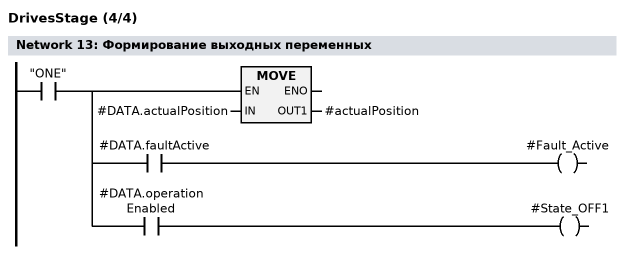
   RUNG wire#powerrail
      Contact( "ONE" )
      wire#w1
      Move(in := #DATA.actualPosition, out1 => #actualPosition)
   END_RUNG
   RUNG wire#w1
      Contact( #DATA.faultActive )
      Coil( #Fault_Active )
   END_RUNG
   RUNG wire#w1
      Contact( #DATA.operationEnabled )
      Coil( #State_OFF1 )
   END_RUNG
   // the same network as SCL:
   IF "ONE" THEN #actualPosition := #DATA.actualPosition; END_IF;
   #Fault_Active := "ONE" AND #DATA.faultActive;
   #State_OFF1 := "ONE" AND #DATA.operationEnabled;
END_REGION
END_FUNCTION_BLOCK

FUNCTION_BLOCK "PD_TEL9_DrivePos"   // FB38011, SCL
TITLE = PD_Tel9_DrivePos
{ S7_Optimized_Access := 'TRUE' }
AUTHOR : SIEMENS
VERSION : 0.1
// Function block to position control a drive using standard telegram 9
   VAR_INPUT
      on : Bool;   // 1 = On, 0 = Off (OFF1)
      noCoastStop : Bool := TRUE;   // 1 = No Coast Stop, 0 = Coast Stop (OFF2)
      noQuickStop : Bool := TRUE;   // 1 = No Quick Stop, 0 = Quick Stop (OFF3)
      enableOperation : Bool := TRUE;   // 1 = Enable operation
      rejectTraversingTask : Bool := TRUE;   // 0 = Reject active traversing task
      intermediateStop : Bool := TRUE;   // 0 = Intermediate STOP active traversing task
      acknowledgeError : Bool;   // Acknowledge faults (0 -> 1)
      jog1 : Bool;   // Jog 1 signal
      jog2 : Bool;   // Jog 2 signal
      startHomingProcedure : Bool;   // Start homing procedure
      activateTraversingTask : Bool;   // Start Traversing for MDI / Traversing Block (0->1 edge) / Activate traversing task
      traversingTaskSelection : UInt;   // Select traversing task (0..1023)
      submode : Bool;   // MDI Activation Signal (1 = MDI activation) / Submode: 0 = program, 1 = MDI
      stw2 : Word;   // Control word 2 (STW2)
      targetPositionMDI : DInt;   // Position Setpoint MDI [LU] / MDI target position
      velocityMDI : DInt;   // Velocity MDI [1000 LU/min] / MDI velocity
      accelerationOverrideMDI : Real := 100.0;   // Acceleration Override MDI (0.1% .. 100.0%) / MDI override of acceleration [%]
      decelerationOverrideMDI : Real := 100.0;   // Deceleration Override MDI (0.1% .. 100.0%) / MDI override of deceleration [%]
      positioningModeMDI : Bool;   // Positioning Type MDI (0 = relative; 1 = absolute) / Positioning mode: 0 = relative, 1 = absolute
      directionPositiveMDI : Bool;   // MDI Positive Positioning Direction / Modulo axis: Absolute positioning in positive direction. If directionPosMDI = directionNegMDI positioning via shortest way.
      directionNegativeMDI : Bool;   // MDI Negative Positioning Direction / Modulo axis: Absolute positioning in negative direction. If directionNegMDI = directionPosMDI positioning via shortest way.
      hardwareId : Hw_Io;   // Hardware identifer of the drive axis
   END_VAR
   VAR_OUTPUT
      operationEnabled : Bool;   // Operation enabled
      switchingOnInhibited : Bool;   // Switching on inhibited
      faultActive : Bool;   // Fault present
      warningActive : Bool;   // Warning present
      homePositionSet : Bool;   // Home position set (axis homed)
      targetPositionReached : Bool;   // Target position reached
      driveStopped : Bool;   // A traversing task has been completed or standstill for intermediate stop
      traversingTaskAcknowledged : Bool;   // A new traversing task or MDI setpoint was started
      actualPosition : DInt;   // Actual position
      activeTraversingTask : UInt;   // Active traversing task
      zsw1 : Word;   // Status word 1
      zsw2 : Word;   // Status word 2
      error : Bool;   // Error active, check status and diagId
      status : Word;   // Status output (7002 = FB in operation; 8xxx = error description - read the manual)
      diagId : DWord;   // Error codes of the cyclic system function blocks GETIO / SETIO
   END_VAR
   VAR
      statError : Bool;   // Static value for output error
      statStatus : Word;   // Static value for output status
      statDiagId : DWord;   // Static value for output diagId
      statCycWrite : Struct   // Structure representing the send direction (PLC to drive) of standard telegram 9
         STW1 : Struct
            jog1 : Bool;   // p2589 EPOS jog 1 signal source
            jog2 : Bool;   // p2590 EPOS jog 2 signal source
            controlByPlc : Bool := TRUE;   // p854[0] Control by PLC/no control by PLC
            homing : Bool;   // p2595 EPOS referencing start
            noDefine1 : Bool;
            externalBlockchange : Bool;   // p2633 EPOS external block change (0 -> 1)
            noDefine2 : Bool;
            noDefine3 : Bool;
            on : Bool;   // p840[0] ON / OFF (OFF1)
            noCoastStop : Bool := TRUE;   // p844[0] No coast-down / coast-down (OFF2) signal source 1
            noQuickStop : Bool := TRUE;   // p848[0] No Quick Stop / Quick Stop (OFF3) signal source 1
            enableOperation : Bool := TRUE;   // p852[0] Enable operation/inhibit operation
            rejectTraversingTask : Bool;   // p2641 EPOS reject traversing task (0 signal)
            intermediateStop : Bool;   // p2640 EPOS intermediate stop (0 signal)
            activateTraversing : Bool;   // p2631 EPOS activate traversing task (0 -> 1)
            acknowledgeFault : Bool;   // p2103[0] Acknowledge faults
         END_STRUCT;
         SATZANW : Struct
            travTaskBit8 : Bool;
            travTaskBit9 : Bool;
            reserve10 : Bool;
            reserve11 : Bool;
            reserve12 : Bool;
            reserve13 : Bool;
            reserve14 : Bool;
            subMode : Bool;
            travTaskBit0 : Bool;
            travTaskBit1 : Bool;
            travTaskBit2 : Bool;
            travTaskBit3 : Bool;
            travTaskBit4 : Bool;
            travTaskBit5 : Bool;
            travTaskBit6 : Bool;
            travTaskBit7 : Bool;
         END_STRUCT;
         STW2 : Struct
            noDefine7 : Bool;
            noDefine8 : Bool;
            noDefine9 : Bool;
            MotorChangeoverFeedback : Bool;   // p828[0] Motor changeover feedback signal
            noDefine10 : Bool;
            noDefine11 : Bool;
            noDefine12 : Bool;
            noDefine13 : Bool;
            DDSSetSelectionBit0 : Bool;   // p820[0] Drive Data Set selection DDS bit 0
            noDefine1 : Bool;
            noDefine2 : Bool;
            noDefine3 : Bool;
            noDefine4 : Bool;
            noDefine5 : Bool;
            noDefine6 : Bool;
            ParkingAxisSelection : Bool;   // p897 Parking axis selection
         END_STRUCT;
         MDI_TARPOS : DInt;
         MDI_VELOCITY : DInt;
         MDI_ACC : UInt;
         MDI_DEC : UInt;
         MDI_MOD : Word;
      END_STRUCT;
      statCycRead : Struct   // Structure representing the receiving direction (PLC from drive) of standard telegram 9
         ZSW1 : Struct
            followingErrorInTolerance : Bool;   // r2684.8 Following error in tolerance
            controlRequest : Bool;   // r899.9 Control request
            targetPosReached : Bool;   // r2684.10 Target position reached
            homePosSet : Bool;   // r2684.11 Reference point set
            acknowledgeTraversingBlockActivated : Bool;   // r2684.12 Acknowledgement traversing block activated
            driveStopped : Bool;   // r2199.0 |n_act| < speed threshold value 3
            setZero1 : Bool;   // r2080.14=0
            setZero2 : Bool;   // r2080.15=0
            readyForSwitchOn : Bool;   // r899.0 Ready for switching on
            ready : Bool;   // r899.1 Ready
            operationEnabled : Bool;   // r899.2 Operation enabled
            faultPresent : Bool;   // r2139.3 Fault present
            noCoastingActive : Bool;   // r899.4 OFF2 active
            noQuickStopActive : Bool;   // r899.5 OFF3 active
            switchingOnInhibitedActive : Bool;   // r899.6 Switching on inhibited active
            warningActive : Bool;   // r2139.7 Alarm present
         END_STRUCT;
         AKTSATZ : Word;
         ZSW2 : Struct
            TravelFixetStopActive : Bool;   // r1406.8 Travel to fixed stop active
            noDefine1 : Bool;
            PulseEnable : Bool;   // r899.11 Pulses enabled
            motorChanghoverActive : Bool;   // r835.0 Motor changeover active
            noDefine2 : Bool;
            noDefine3 : Bool;
            noDefine4 : Bool;
            noDefine5 : Bool;
            DataSetBit0 : Bool;   // r51.0 Drive Data Set DDS effective bit 0
            DataSetBit1 : Bool;   // r51.1 Drive Data Set DDS effective bit 1
            noDefine6 : Bool;
            noDefine7 : Bool;
            noDefine8 : Bool;
            AlarmclassBit0 : Bool;   // r2139.11 Alarm class bit 0
            AlarmclassBit1 : Bool;   // r2139.12 Alarm class bit 1
            ParkingAxisActive : Bool;   // r896.0 Parking axis active
         END_STRUCT;
         XIST_A : DInt;
      END_STRUCT;
   END_VAR
   VAR_TEMP
      tempSendBuffer : Array[0..9] of Word;   // Buffer to write to the drive
      tempReadBuffer : Array[0..4] of Word;   // Buffer to read from the drive
      tempRetGETIO : DWord;   // Status of GETIO command
      tempRetSETIO : DWord;   // Status of SETIO command
      tempDWord : DWord;   // Temporary Dword for calculations
      tempReal : Real;   // Temporary Real for calculations
   END_VAR
   VAR CONSTANT
      MAX_INT : Int := 16#7FFF;   // 7FFFh = +200%
      MIN_INT : Int := 16#0;   // 0h = 0%
      NORMALIZATION_REAL : Real := 163.84;
      TRAVERSE_TASK_LIMIT : UInt := 2#1111111111;   // Maximum 1024 traversing tasks are allowed
      STATUS_IN_OPERATION : Word := 16#7002;   // FB is in operation
      ERROR_INVALID_TRV_TASK : Word := 16#8204;   // Invalid traversing task selected, choose a valid traversing task from 0 to 1023
      ERROR_DRIVE_ERROR : Word := 16#8401;   // Drive has error
      ERROR_SWITCH_ON_INHIBITED : Word := 16#8402;   // Switch on inhibited by the drive
      ERROR_SETIO : Word := 16#8600;   // Error occured when writing telegram data (SETIO command)
      ERROR_GETIO : Word := 16#8601;   // Error occured when reading telegram data (GETIO command)
   END_VAR
BEGIN
   //=============================================================================
   //SIEMENS AG
   //(c)Copyright 2019 All Rights Reserved
   //-----------------------------------------------------------------------------
   //Library: -
   //Tested with: SIMATIC S7-1513-1 PN V2.6 and SINAMICS S120 CU320-2 PN V5.2 HF1
   //Engineering: TIA Portal V15.1
   //Restrictions: -
   //Requirements: Drive supporting PROFIdrive standard telegram 9
   //Functionality: Function block to position control a drive using PROFIdrive standard telegram 9
   //-----------------------------------------------------------------------------
   //Change log table:
   //Version  Date       Expert in charge Changes applied
   //01.00.00 03.12.2019 (AS) First released version
   //=============================================================================

   REGION ResetFbState
       #statError := FALSE;
       #statDiagId := 16#0;
       #statStatus := #STATUS_IN_OPERATION;
   END_REGION

   REGION ReadCyclicData    
       //Read cyclic telegram data
       "GETIO_DB"(ID := #hardwareId,
                  STATUS => #tempRetGETIO,
                  INPUTS := #tempReadBuffer);

       // write GETIO status to diagId

       #tempRetGETIO := SHR(IN := #tempRetGETIO, N := 8);
       #tempRetGETIO := #tempRetGETIO & 16#FFFF;

       IF #tempRetGETIO <> 0 THEN
           #statStatus := #ERROR_GETIO;
           #statDiagId := #tempRetGETIO;
       END_IF;
   END_REGION

   REGION CopyReadValuesToStatData
       //copy all values from read temp array to static data
       #statCycRead.ZSW1.followingErrorInTolerance := #tempReadBuffer[0].%X8;
       #statCycRead.ZSW1.controlRequest := #tempReadBuffer[0].%X9;
       #statCycRead.ZSW1.targetPosReached := #tempReadBuffer[0].%X10;
       #statCycRead.ZSW1.homePosSet := #tempReadBuffer[0].%X11;
       #statCycRead.ZSW1.acknowledgeTraversingBlockActivated := #tempReadBuffer[0].%X12;
       #statCycRead.ZSW1.driveStopped := #tempReadBuffer[0].%X13;
       #statCycRead.ZSW1.setZero1 := #tempReadBuffer[0].%X14;
       #statCycRead.ZSW1.setZero2 := #tempReadBuffer[0].%X15;
       #statCycRead.ZSW1.readyForSwitchOn := #tempReadBuffer[0].%X0;
       #statCycRead.ZSW1.ready := #tempReadBuffer[0].%X1;
       #statCycRead.ZSW1.operationEnabled := #tempReadBuffer[0].%X2;
       #statCycRead.ZSW1.faultPresent := #tempReadBuffer[0].%X3;
       #statCycRead.ZSW1.noCoastingActive := #tempReadBuffer[0].%X4;
       #statCycRead.ZSW1.noQuickStopActive := #tempReadBuffer[0].%X5;
       #statCycRead.ZSW1.switchingOnInhibitedActive := #tempReadBuffer[0].%X6;
       #statCycRead.ZSW1.warningActive := #tempReadBuffer[0].%X7;

       #statCycRead.ZSW2.TravelFixetStopActive := #tempReadBuffer[2].%X8;
       #statCycRead.ZSW2.noDefine1 := #tempReadBuffer[2].%X9;
       #statCycRead.ZSW2.PulseEnable := #tempReadBuffer[2].%X10;
       #statCycRead.ZSW2.motorChanghoverActive := #tempReadBuffer[2].%X11;
       #statCycRead.ZSW2.noDefine2 := #tempReadBuffer[2].%X12;
       #statCycRead.ZSW2.noDefine3 := #tempReadBuffer[2].%X13;
       #statCycRead.ZSW2.noDefine4 := #tempReadBuffer[2].%X14;
       #statCycRead.ZSW2.noDefine5 := #tempReadBuffer[2].%X15;
       #statCycRead.ZSW2.DataSetBit0 := #tempReadBuffer[2].%X0;
       #statCycRead.ZSW2.DataSetBit1 := #tempReadBuffer[2].%X1;
       #statCycRead.ZSW2.noDefine6 := #tempReadBuffer[2].%X2;
       #statCycRead.ZSW2.noDefine7 := #tempReadBuffer[2].%X3;
       #statCycRead.ZSW2.noDefine8 := #tempReadBuffer[2].%X4;
       #statCycRead.ZSW2.AlarmclassBit0 := #tempReadBuffer[2].%X5;
       #statCycRead.ZSW2.AlarmclassBit1 := #tempReadBuffer[2].%X6;
       #statCycRead.ZSW2.ParkingAxisActive := #tempReadBuffer[2].%X7;

       #statCycRead.AKTSATZ := #tempReadBuffer[1];

       #statCycRead.XIST_A.%W0 := #tempReadBuffer[4];
       #statCycRead.XIST_A.%W1 := #tempReadBuffer[3];
   END_REGION

   REGION WriteOutputs    
       // write status from telegram to block outputs
       #operationEnabled := #statCycRead.ZSW1.operationEnabled;
       #switchingOnInhibited := #statCycRead.ZSW1.switchingOnInhibitedActive;
       #faultActive := #statCycRead.ZSW1.faultPresent;
       #warningActive := #statCycRead.ZSW1.warningActive;
       #homePositionSet := #statCycRead.ZSW1.homePosSet;
       #targetPositionReached := #statCycRead.ZSW1.targetPosReached;
       #driveStopped := #statCycRead.ZSW1.driveStopped;
       #traversingTaskAcknowledged := #statCycRead.ZSW1.acknowledgeTraversingBlockActivated;
       #actualPosition := #statCycRead.XIST_A;
       #activeTraversingTask := WORD_TO_UINT(#statCycRead.AKTSATZ);
       #zsw1 := #tempReadBuffer[0];
       #zsw2 := #tempReadBuffer[2];
   END_REGION

   REGION ReadInputs    
       #statCycWrite.STW1.on := #on;
       #statCycWrite.STW1.noCoastStop := #noCoastStop;
       #statCycWrite.STW1.noQuickStop := #noQuickStop;
       #statCycWrite.STW1.rejectTraversingTask := #rejectTraversingTask;
       #statCycWrite.STW1.intermediateStop := #intermediateStop;
       #statCycWrite.STW1.acknowledgeFault := #acknowledgeError;
       #statCycWrite.STW1.jog1 := #jog1;
       #statCycWrite.STW1.jog2 := #jog2;
       #statCycWrite.STW1.homing := #startHomingProcedure;
       #statCycWrite.STW1.activateTraversing := #activateTraversingTask;

       #statCycWrite.SATZANW.travTaskBit0 := #traversingTaskSelection.%X0;
       #statCycWrite.SATZANW.travTaskBit1 := #traversingTaskSelection.%X1;
       #statCycWrite.SATZANW.travTaskBit2 := #traversingTaskSelection.%X2;
       #statCycWrite.SATZANW.travTaskBit3 := #traversingTaskSelection.%X3;
       #statCycWrite.SATZANW.travTaskBit4 := #traversingTaskSelection.%X4;
       #statCycWrite.SATZANW.travTaskBit5 := #traversingTaskSelection.%X5;
       #statCycWrite.SATZANW.travTaskBit6 := #traversingTaskSelection.%X6;
       #statCycWrite.SATZANW.travTaskBit7 := #traversingTaskSelection.%X7;
       #statCycWrite.SATZANW.travTaskBit8 := #traversingTaskSelection.%X8;
       #statCycWrite.SATZANW.travTaskBit9 := #traversingTaskSelection.%X9;
       #statCycWrite.SATZANW.subMode := #submode;

       #statCycWrite.STW2.DDSSetSelectionBit0 := #stw2.%X0;
       #statCycWrite.STW2.noDefine1 := #stw2.%X1;
       #statCycWrite.STW2.noDefine2 := #stw2.%X2;
       #statCycWrite.STW2.noDefine3 := #stw2.%X3;
       #statCycWrite.STW2.noDefine4 := #stw2.%X4;
       #statCycWrite.STW2.noDefine5 := #stw2.%X5;
       #statCycWrite.STW2.noDefine6 := #stw2.%X6;
       #statCycWrite.STW2.ParkingAxisSelection := #stw2.%X7;
       #statCycWrite.STW2.noDefine7 := #stw2.%X8;
       #statCycWrite.STW2.noDefine8 := #stw2.%X9;
       #statCycWrite.STW2.noDefine9 := #stw2.%X10;
       #statCycWrite.STW2.MotorChangeoverFeedback := #stw2.%X11;
       #statCycWrite.STW2.noDefine10 := #stw2.%X12;
       #statCycWrite.STW2.noDefine11 := #stw2.%X13;
       #statCycWrite.STW2.noDefine12 := #stw2.%X14;
       #statCycWrite.STW2.noDefine13 := #stw2.%X15;

       #statCycWrite.MDI_TARPOS := #targetPositionMDI;
       #statCycWrite.MDI_VELOCITY := #velocityMDI;

       #tempReal := #accelerationOverrideMDI * #NORMALIZATION_REAL;
       // Limit REAL - Variable to INT - limits
       IF #tempReal > #MAX_INT THEN
           #tempReal := #MAX_INT;
       ELSIF #tempReal < #MIN_INT THEN
           #tempReal := #MIN_INT;
       ELSE
           ; // not needed
       END_IF;
       #statCycWrite.MDI_ACC := INT_TO_WORD(REAL_TO_INT(#tempReal));

       #tempReal := #decelerationOverrideMDI * #NORMALIZATION_REAL;
       // Limit REAL - Variable to INT - limits
       IF #tempReal > #MAX_INT THEN
           #tempReal := #MAX_INT;
       ELSIF #tempReal < #MIN_INT THEN
           #tempReal := #MIN_INT;
       ELSE
           ; // not needed
       END_IF;
       #statCycWrite.MDI_DEC := INT_TO_WORD(REAL_TO_INT(#tempReal));

       //MDI_MODE (bitwise inputs to word)
       #statCycWrite.MDI_MOD.%X0 := #positioningModeMDI;
       #statCycWrite.MDI_MOD.%X1 := #directionPositiveMDI;
       #statCycWrite.MDI_MOD.%X2 := #directionNegativeMDI;

       IF #traversingTaskSelection > #TRAVERSE_TASK_LIMIT THEN
           #statStatus := #ERROR_INVALID_TRV_TASK;
       END_IF;
   END_REGION

   REGION CopyWriteValuesToTempArray
       //copy all cyclic data from stat data to temp array
       #tempSendBuffer[0].%X0 := #statCycWrite.STW1.on;
       #tempSendBuffer[0].%X1 := #statCycWrite.STW1.noCoastStop;
       #tempSendBuffer[0].%X2 := #statCycWrite.STW1.noQuickStop;
       #tempSendBuffer[0].%X3 := #statCycWrite.STW1.enableOperation;
       #tempSendBuffer[0].%X4 := #statCycWrite.STW1.rejectTraversingTask;
       #tempSendBuffer[0].%X5 := #statCycWrite.STW1.intermediateStop;
       #tempSendBuffer[0].%X6 := #statCycWrite.STW1.activateTraversing;
       #tempSendBuffer[0].%X7 := #statCycWrite.STW1.acknowledgeFault;
       #tempSendBuffer[0].%X8 := #statCycWrite.STW1.jog1;
       #tempSendBuffer[0].%X9 := #statCycWrite.STW1.jog2;
       #tempSendBuffer[0].%X10 := #statCycWrite.STW1.controlByPlc;
       #tempSendBuffer[0].%X11 := #statCycWrite.STW1.homing;
       #tempSendBuffer[0].%X12 := #statCycWrite.STW1.noDefine1;
       #tempSendBuffer[0].%X13 := #statCycWrite.STW1.externalBlockchange;
       #tempSendBuffer[0].%X14 := #statCycWrite.STW1.noDefine2;
       #tempSendBuffer[0].%X15 := #statCycWrite.STW1.noDefine3;

       #tempSendBuffer[1].%X0 := #statCycWrite.SATZANW.travTaskBit0;
       #tempSendBuffer[1].%X1 := #statCycWrite.SATZANW.travTaskBit1;
       #tempSendBuffer[1].%X2 := #statCycWrite.SATZANW.travTaskBit2;
       #tempSendBuffer[1].%X3 := #statCycWrite.SATZANW.travTaskBit3;
       #tempSendBuffer[1].%X4 := #statCycWrite.SATZANW.travTaskBit4;
       #tempSendBuffer[1].%X5 := #statCycWrite.SATZANW.travTaskBit5;
       #tempSendBuffer[1].%X6 := #statCycWrite.SATZANW.travTaskBit6;
       #tempSendBuffer[1].%X7 := #statCycWrite.SATZANW.travTaskBit7;
       #tempSendBuffer[1].%X8 := #statCycWrite.SATZANW.travTaskBit8;
       #tempSendBuffer[1].%X9 := #statCycWrite.SATZANW.travTaskBit9;
       #tempSendBuffer[1].%X10 := #statCycWrite.SATZANW.reserve10;
       #tempSendBuffer[1].%X11 := #statCycWrite.SATZANW.reserve11;
       #tempSendBuffer[1].%X12 := #statCycWrite.SATZANW.reserve12;
       #tempSendBuffer[1].%X13 := #statCycWrite.SATZANW.reserve13;
       #tempSendBuffer[1].%X14 := #statCycWrite.SATZANW.reserve14;
       #tempSendBuffer[1].%X15 := #statCycWrite.SATZANW.subMode;

       #tempSendBuffer[2].%X0 := #statCycWrite.STW2.DDSSetSelectionBit0;
       #tempSendBuffer[2].%X1 := #statCycWrite.STW2.noDefine1;
       #tempSendBuffer[2].%X2 := #statCycWrite.STW2.noDefine2;
       #tempSendBuffer[2].%X3 := #statCycWrite.STW2.noDefine3;
       #tempSendBuffer[2].%X4 := #statCycWrite.STW2.noDefine4;
       #tempSendBuffer[2].%X5 := #statCycWrite.STW2.noDefine5;
       #tempSendBuffer[2].%X6 := #statCycWrite.STW2.noDefine6;
       #tempSendBuffer[2].%X7 := #statCycWrite.STW2.ParkingAxisSelection;
       #tempSendBuffer[2].%X8 := #statCycWrite.STW2.noDefine7;
       #tempSendBuffer[2].%X9 := #statCycWrite.STW2.noDefine8;
       #tempSendBuffer[2].%X10 := #statCycWrite.STW2.noDefine9;
       #tempSendBuffer[2].%X11 := #statCycWrite.STW2.MotorChangeoverFeedback;
       #tempSendBuffer[2].%X12 := #statCycWrite.STW2.noDefine10;
       #tempSendBuffer[2].%X13 := #statCycWrite.STW2.noDefine11;
       #tempSendBuffer[2].%X14 := #statCycWrite.STW2.noDefine12;
       #tempSendBuffer[2].%X15 := #statCycWrite.STW2.noDefine13;

       #tempDWord := DINT_TO_DWORD(#statCycWrite.MDI_TARPOS);
       #tempSendBuffer[3] := #tempDWord.%W1;
       #tempSendBuffer[4] := #tempDWord.%W0;

       #tempDWord := DINT_TO_DWORD(#statCycWrite.MDI_VELOCITY);
       #tempSendBuffer[5] := #tempDWord.%W1;
       #tempSendBuffer[6] := #tempDWord.%W0;

       #tempSendBuffer[7] := #statCycWrite.MDI_ACC;
       #tempSendBuffer[8] := #statCycWrite.MDI_DEC;
       #tempSendBuffer[9] := #statCycWrite.MDI_MOD;
   END_REGION

   REGION WriteCyclicData
       //Write cyclic telegram data
       "SETIO_DB"(ID:=#hardwareId,
                  STATUS=>#tempRetSETIO,
                  OUTPUTS:=#statCycWrite);

       // write SETIO status to diagId
       #tempRetSETIO:=SHR(IN := #tempRetSETIO, N := 8);
       #tempRetSETIO := #tempRetSETIO & 16#FFFF;

       IF #tempRetSETIO <> 0 THEN
           #statStatus := #ERROR_SETIO;
           #statDiagId := #tempRetSETIO;
       END_IF;
   END_REGION

   REGION ErrorHandling
       IF #faultActive THEN
           #statStatus := #ERROR_DRIVE_ERROR;
       END_IF;

       IF #switchingOnInhibited THEN
           #statStatus := #ERROR_SWITCH_ON_INHIBITED;
       END_IF;

       // set error output
       IF #statDiagId <> 0 OR #statStatus <> #STATUS_IN_OPERATION THEN
           #statError := TRUE;
       ELSE
           #statError := FALSE;
       END_IF;
   END_REGION

   REGION WriteOutputs
       #error := #statError;
       #status := #statStatus;
       #diagId := #statDiagId;
   END_REGION
END_FUNCTION_BLOCK

FUNCTION "StateMachineDRIVE" : Void   // FC5, LAD
{ S7_Optimized_Access := 'TRUE' }
VERSION : 0.1
   VAR_TEMP
      disIRT_count : Int;
      enIRT_count : Int;
   END_VAR
BEGIN

REGION Network 1 (SCL): Привод 1 и 2
   // Первый привод. 
   "TEL9_Drive1".OFF2 := TRUE;
   "TEL9_Drive1".OFF3 := TRUE;
   "TEL9_Drive1".enableOperation := TRUE;
   "TEL9_Drive1".directionPositiveMDI := TRUE;
   // Второй привод. 
   "TEL9_Drive2".OFF2 := TRUE;
   "TEL9_Drive2".OFF3 := TRUE;
   "TEL9_Drive2".enableOperation := TRUE;
   "TEL9_Drive2".directionPositiveMDI := TRUE;
END_REGION

REGION Network 2: Работа с первым приводом
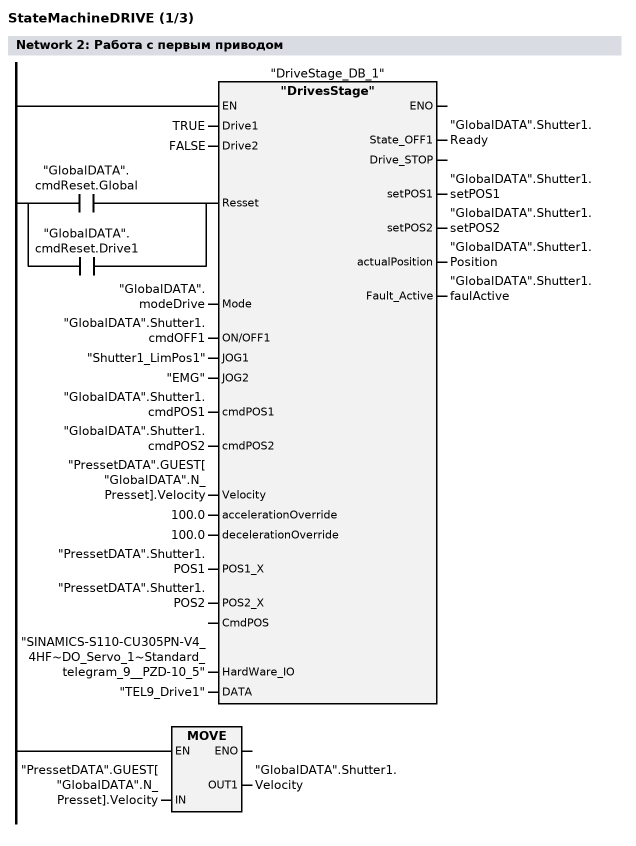
   RUNG wire#powerrail
      "DriveStage_DB_1"(Resset := wire#w1, Drive1 := TRUE, Drive2 := FALSE, Mode := "GlobalDATA".modeDrive, "ON/OFF1" := "GlobalDATA".Shutter1.cmdOFF1, JOG1 := "Shutter1_LimPos1", JOG2 := "EMG", cmdPOS1 := "GlobalDATA".Shutter1.cmdPOS1, cmdPOS2 := "GlobalDATA".Shutter1.cmdPOS2, Velocity := "PressetDATA".GUEST["GlobalDATA".N_Presset].Velocity, accelerationOverride := 100.0, decelerationOverride := 100.0, POS1_X := "PressetDATA".Shutter1.POS1, POS2_X := "PressetDATA".Shutter1.POS2, CmdPOS :=, HardWare_IO := "SINAMICS-S110-CU305PN-V4_4HF~DO_Servo_1~Standard_telegram_9__PZD-10_5", DATA := "TEL9_Drive1", State_OFF1 => "GlobalDATA".Shutter1.Ready, Drive_STOP =>, setPOS1 => "GlobalDATA".Shutter1.setPOS1, setPOS2 => "GlobalDATA".Shutter1.setPOS2, actualPosition => "GlobalDATA".Shutter1.Position, Fault_Active => "GlobalDATA".Shutter1.faulActive)
   END_RUNG
   RUNG wire#powerrail
      Contact( "GlobalDATA".cmdReset.Global )
   END_RUNG wire#w1
   RUNG wire#powerrail
      Contact( "GlobalDATA".cmdReset.Drive1 )
   END_RUNG wire#w1
   RUNG wire#powerrail
      Move(in := "PressetDATA".GUEST["GlobalDATA".N_Presset].Velocity, out1 => "GlobalDATA".Shutter1.Velocity)
   END_RUNG
   // the same network as SCL:
   "DriveStage_DB_1"(Drive1 := TRUE,   // "DrivesStage"
                     Drive2 := FALSE,
                     Resset := "GlobalDATA".cmdReset.Global OR "GlobalDATA".cmdReset.Drive1,
                     Mode := "GlobalDATA".modeDrive,
                     "ON/OFF1" := "GlobalDATA".Shutter1.cmdOFF1,
                     JOG1 := "Shutter1_LimPos1",
                     JOG2 := "EMG",
                     cmdPOS1 := "GlobalDATA".Shutter1.cmdPOS1,
                     cmdPOS2 := "GlobalDATA".Shutter1.cmdPOS2,
                     Velocity := "PressetDATA".GUEST["GlobalDATA".N_Presset].Velocity,
                     accelerationOverride := 100.0,
                     decelerationOverride := 100.0,
                     POS1_X := "PressetDATA".Shutter1.POS1,
                     POS2_X := "PressetDATA".Shutter1.POS2,
                     HardWare_IO := "SINAMICS-S110-CU305PN-V4_4HF~DO_Servo_1~Standard_telegram_9__PZD-10_5",
                     DATA := "TEL9_Drive1",
                     State_OFF1 => "GlobalDATA".Shutter1.Ready,
                     setPOS1 => "GlobalDATA".Shutter1.setPOS1,
                     setPOS2 => "GlobalDATA".Shutter1.setPOS2,
                     actualPosition => "GlobalDATA".Shutter1.Position,
                     Fault_Active => "GlobalDATA".Shutter1.faulActive);
   "GlobalDATA".Shutter1.Velocity := "PressetDATA".GUEST["GlobalDATA".N_Presset].Velocity;
END_REGION

REGION Network 3: Работа со вторым приводом
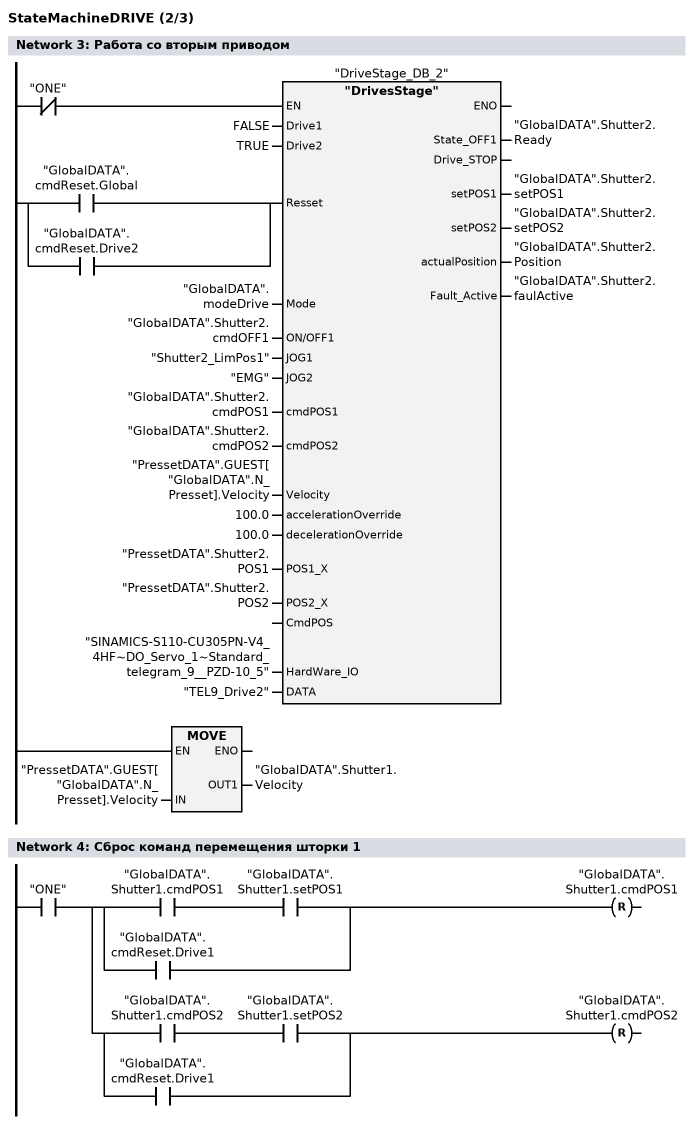
   RUNG wire#powerrail
      I_Contact( "ONE" )
      "DriveStage_DB_2"(Resset := wire#w1, Drive1 := FALSE, Drive2 := TRUE, Mode := "GlobalDATA".modeDrive, "ON/OFF1" := "GlobalDATA".Shutter2.cmdOFF1, JOG1 := "Shutter2_LimPos1", JOG2 := "EMG", cmdPOS1 := "GlobalDATA".Shutter2.cmdPOS1, cmdPOS2 := "GlobalDATA".Shutter2.cmdPOS2, Velocity := "PressetDATA".GUEST["GlobalDATA".N_Presset].Velocity, accelerationOverride := 100.0, decelerationOverride := 100.0, POS1_X := "PressetDATA".Shutter2.POS1, POS2_X := "PressetDATA".Shutter2.POS2, CmdPOS :=, HardWare_IO := "SINAMICS-S110-CU305PN-V4_4HF~DO_Servo_1~Standard_telegram_9__PZD-10_5", DATA := "TEL9_Drive2", State_OFF1 => "GlobalDATA".Shutter2.Ready, Drive_STOP =>, setPOS1 => "GlobalDATA".Shutter2.setPOS1, setPOS2 => "GlobalDATA".Shutter2.setPOS2, actualPosition => "GlobalDATA".Shutter2.Position, Fault_Active => "GlobalDATA".Shutter2.faulActive)
   END_RUNG
   RUNG wire#powerrail
      Contact( "GlobalDATA".cmdReset.Global )
   END_RUNG wire#w1
   RUNG wire#powerrail
      Contact( "GlobalDATA".cmdReset.Drive2 )
   END_RUNG wire#w1
   RUNG wire#powerrail
      Move(in := "PressetDATA".GUEST["GlobalDATA".N_Presset].Velocity, out1 => "GlobalDATA".Shutter1.Velocity)
   END_RUNG
   // the same network as SCL:
   IF NOT "ONE" THEN
       "DriveStage_DB_2"(Drive1 := FALSE,   // "DrivesStage"
                         Drive2 := TRUE,
                         Resset := "GlobalDATA".cmdReset.Global OR "GlobalDATA".cmdReset.Drive2,
                         Mode := "GlobalDATA".modeDrive,
                         "ON/OFF1" := "GlobalDATA".Shutter2.cmdOFF1,
                         JOG1 := "Shutter2_LimPos1",
                         JOG2 := "EMG",
                         cmdPOS1 := "GlobalDATA".Shutter2.cmdPOS1,
                         cmdPOS2 := "GlobalDATA".Shutter2.cmdPOS2,
                         Velocity := "PressetDATA".GUEST["GlobalDATA".N_Presset].Velocity,
                         accelerationOverride := 100.0,
                         decelerationOverride := 100.0,
                         POS1_X := "PressetDATA".Shutter2.POS1,
                         POS2_X := "PressetDATA".Shutter2.POS2,
                         HardWare_IO := "SINAMICS-S110-CU305PN-V4_4HF~DO_Servo_1~Standard_telegram_9__PZD-10_5",
                         DATA := "TEL9_Drive2",
                         State_OFF1 => "GlobalDATA".Shutter2.Ready,
                         setPOS1 => "GlobalDATA".Shutter2.setPOS1,
                         setPOS2 => "GlobalDATA".Shutter2.setPOS2,
                         actualPosition => "GlobalDATA".Shutter2.Position,
                         Fault_Active => "GlobalDATA".Shutter2.faulActive);
   END_IF;
   "GlobalDATA".Shutter1.Velocity := "PressetDATA".GUEST["GlobalDATA".N_Presset].Velocity;
END_REGION

REGION Network 4: Сброс команд перемещения шторки 1
   RUNG wire#powerrail
      Contact( "ONE" )
      wire#w1
      Contact( "GlobalDATA".Shutter1.cmdPOS1 )
      Contact( "GlobalDATA".Shutter1.setPOS1 )
      wire#w2
      R_Coil( "GlobalDATA".Shutter1.cmdPOS1 )
   END_RUNG
   RUNG wire#w1
      Contact( "GlobalDATA".cmdReset.Drive1 )
   END_RUNG wire#w2
   RUNG wire#w1
      Contact( "GlobalDATA".Shutter1.cmdPOS2 )
      Contact( "GlobalDATA".Shutter1.setPOS2 )
      wire#w3
      R_Coil( "GlobalDATA".Shutter1.cmdPOS2 )
   END_RUNG
   RUNG wire#w1
      Contact( "GlobalDATA".cmdReset.Drive1 )
   END_RUNG wire#w3
   // the same network as SCL:
   IF "ONE" AND (("GlobalDATA".Shutter1.cmdPOS1 AND "GlobalDATA".Shutter1.setPOS1) OR "GlobalDATA".cmdReset.Drive1) THEN
       "GlobalDATA".Shutter1.cmdPOS1 := FALSE;
   END_IF;
   IF "ONE" AND (("GlobalDATA".Shutter1.cmdPOS2 AND "GlobalDATA".Shutter1.setPOS2) OR "GlobalDATA".cmdReset.Drive1) THEN
       "GlobalDATA".Shutter1.cmdPOS2 := FALSE;
   END_IF;
END_REGION

REGION Network 5: Сброс команд перемещения шторки 2
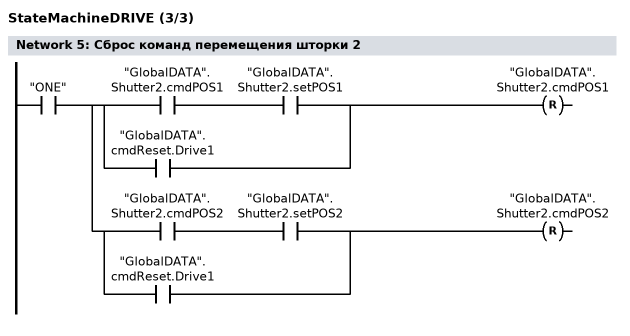
   RUNG wire#powerrail
      Contact( "ONE" )
      wire#w1
      Contact( "GlobalDATA".Shutter2.cmdPOS1 )
      Contact( "GlobalDATA".Shutter2.setPOS1 )
      wire#w2
      R_Coil( "GlobalDATA".Shutter2.cmdPOS1 )
   END_RUNG
   RUNG wire#w1
      Contact( "GlobalDATA".cmdReset.Drive1 )
   END_RUNG wire#w2
   RUNG wire#w1
      Contact( "GlobalDATA".Shutter2.cmdPOS2 )
      Contact( "GlobalDATA".Shutter2.setPOS2 )
      wire#w3
      R_Coil( "GlobalDATA".Shutter2.cmdPOS2 )
   END_RUNG
   RUNG wire#w1
      Contact( "GlobalDATA".cmdReset.Drive1 )
   END_RUNG wire#w3
   // the same network as SCL:
   IF "ONE" AND (("GlobalDATA".Shutter2.cmdPOS1 AND "GlobalDATA".Shutter2.setPOS1) OR "GlobalDATA".cmdReset.Drive1) THEN
       "GlobalDATA".Shutter2.cmdPOS1 := FALSE;
   END_IF;
   IF "ONE" AND (("GlobalDATA".Shutter2.cmdPOS2 AND "GlobalDATA".Shutter2.setPOS2) OR "GlobalDATA".cmdReset.Drive1) THEN
       "GlobalDATA".Shutter2.cmdPOS2 := FALSE;
   END_IF;
END_REGION
END_FUNCTION

FUNCTION "CalcPreset" : Void   // FC12, SCL
{ S7_Optimized_Access := 'TRUE' }
VERSION : 0.1
   VAR_INPUT
      Texposure : UInt;   // ms, Time of exposure
   END_VAR
   VAR_OUTPUT
      Velocity : DInt;   // mm/min, Velocity of shutter
      Ttrigger : Time;   // ms, Trigger time for CareRay
      Error : Bool;   // Error present duiring calculate
   END_VAR
   VAR_TEMP
      Tramp : DInt;
      err : Bool;
      Velo : DInt;
      RampTime : Time;
      ExposureTime : Time;
      TriggerTime : Time;
      X : DInt;
      X1 : DInt;
      X2 : DInt;
      T1 : DInt;
      T2 : DInt;
      T3 : DInt;
   END_VAR
BEGIN
   //Проверяем значение экспозиции на допустимые значения
   IF #Texposure < "TexposureMIN" OR #Texposure > "TexposureMAX" THEN
       #err := TRUE;
   ELSE
       //Производим вычисление скорости перемещения шторки в зависимости от заданного времени экспозиции
       #Velo := "Xexposure" * 60 / #Texposure;
       //Если рассчетная скорость выхе или ниже допустимой, то выдаем ошибку
       IF #Velo < "Velo_min" OR #Velo > "Velo_max"  THEN
           #err := TRUE;
       ELSE
           #X := "PressetDATA".Shutter1.POS2 - "PressetDATA".Shutter1.POS1;
           #X1 := #Velo * #Velo / 2 / "AccShutter";
           #X2 := (#X - 2 * #X1 - "Xexposure") / 2;
           //Вычисляем время разгона и торможения
           #T1 := #Velo * 60 / "AccShutter";
           #T2 := #X2 * 60 / #Velo;
           #T3 := #Texposure + 2 * #T1 + 2 * #T2;
           //Преобразуем значение в формат времени
           #TriggerTime := DINT_TO_TIME(#T3);
       END_IF;
   END_IF;

   //Обновляем выходные параметры
   IF #err= FALSE THEN
       #Velocity := #Velo;
       #Ttrigger := #TriggerTime;
   ELSE
       #Error := TRUE;
   END_IF;
END_FUNCTION

// folder: Generators

FUNCTION_BLOCK "GeneratorWarm"   // FB1, SCL
{ S7_Optimized_Access := 'TRUE' }
VERSION : 0.1
   VAR_INPUT
      enable : Bool;
      reset : Bool;
      DataTable : "typeWarmTable";
      readyGenerator : Bool;
      faultGenerator : Bool;
   END_VAR
   VAR_OUTPUT
      busy : Bool;
      done : Bool;
      fault : Bool;
      TimeOut : Time;
   END_VAR
   VAR_IN_OUT
      table : UInt;
      GeneratorDATA : "typeGeneratorDATA";
      "X-RAY_ON" : Bool;
   END_VAR
   VAR
      statStageWarm : UInt;
      statOldStageWarm : UInt;
      statTime : Time;
      statTimeOveral : Time;
      statTimeOff : Time;
      statOldEnable : Bool;
      statTimeStageEn : Bool;
      statStageDone : Bool;
      statOldStage : Bool;
      statVP_done : Bool;
      statCP_done : Bool;
      statCMDUpdate : Bool;
      statTimeBrakeWarm : Bool;
      statTimeBrakeEN : Bool;
      statBrakeWarm : Bool;
      statFault : Bool;
   END_VAR
BEGIN
   IF (#enable = FALSE AND #statOldEnable = TRUE AND #statStageWarm <> 0 AND #"X-RAY_ON" = TRUE)
       OR #table = 0
       OR #reset = TRUE
       OR #enable = FALSE THEN
       #statStageWarm := 0;
       #statStageDone := FALSE;
      // #"X-RAY_ON" := FALSE;
       #table := 0;
       #statTimeStageEn := FALSE;
       #statTimeOveral := T#0ms;
       #busy := FALSE;
       #fault := FALSE;
       #statTimeStageEn := 0;
       #statTimeBrakeEN := 0;
       #TimeOut := T#0s;
       #statFault := FALSE;
   END_IF;

   #statOldEnable := #enable;

   //Проверяем пришел ли новый запрос на прогрев гененератора
   IF (#table > 0)
       AND (#table < 4)
       AND #enable = TRUE
       AND #statOldStageWarm = 0
   THEN
       #statStageDone := TRUE;
       #statTime := #DataTable.T[#table];
       #statTimeOveral := #statTime * 10;
       #busy := TRUE;
       #statStageWarm := 1;
   ELSIF #table = 0 THEN
       #statStageWarm := 0;
       #statStageDone := FALSE;
       #busy := FALSE;
       #statTimeStageEn := 0;
       #statTimeBrakeEN := 0;
       #TimeOut:= T#0s;
   END_IF;



   IF #statStageDone = TRUE THEN
       #statStageDone := FALSE;
       #statTimeStageEn := FALSE;

       #GeneratorDATA.VP_Programm := #DataTable.VP[#statStageWarm];
       #GeneratorDATA.CP_Programm := #DataTable.CP[#statStageWarm];
       #GeneratorDATA.CMD_VP := TRUE;
       #GeneratorDATA.CMD_CP := TRUE;
       #statVP_done := FALSE;
       #statCP_done := FALSE;
   END_IF;

   #statOldStageWarm := #statStageWarm;

   // Проверка выполнения команды по установке напряжения генератора
   IF  #GeneratorDATA.cmdDone = TRUE AND #GeneratorDATA.cmd_Nunmber = "cmdSVLT"  THEN
       #statVP_done := TRUE;
   END_IF;

   // Проверка выполнения команды по установке тока генератора
   IF #GeneratorDATA.cmdDone = TRUE AND #GeneratorDATA.cmd_Nunmber = "cmdSCUR" THEN
       #statCP_done := TRUE;
   END_IF;

   // Проверка установленного значения напряжения и тока
   IF #statCP_done = TRUE AND #statVP_done = TRUE THEN
       #statTimeStageEn := TRUE;
   ELSE
       #statTimeStageEn := FALSE;
   END_IF;

   //Разрешение на проверку тайминга на выполнение команды
   IF (#GeneratorDATA.CMD_VP = TRUE OR #GeneratorDATA.CMD_CP=TRUE) THEN
       // Statement section IF
       #statTimeBrakeEN := TRUE;
       #"X-RAY_ON" := TRUE;
   ELSE
       #statTimeBrakeEN := FALSE;
   END_IF;
   (*
   // Если превышен тайминг между выполнением команд установки напряжения и тока или ошибка генератора, то прерываем процесс прогрева
   IF #faultGenerator = TRUE
       OR #statTimeBrakeWarm = TRUE
       OR #readyGenerator = FALSE
   THEN
       #statBrakeWarm := TRUE;
   ELSE
       #statBrakeWarm := FALSE;
   END_IF;
   *)
   // Отключаем X-RAY, завершаем процесс прогрева
   IF #statBrakeWarm = TRUE
       OR #reset = TRUE
       OR (#statStageWarm >= 11)
       OR #faultGenerator = TRUE
       OR #statFault = TRUE
   THEN
       #statStageWarm := 0;
       #statStageDone := FALSE;
       #"X-RAY_ON" := FALSE;
       #table := 0;
       #done := TRUE;
       #fault := FALSE;
       #busy := FALSE;
   END_IF;

   //Обновляем выходные переменные
   IF #statBrakeWarm = TRUE
       OR #faultGenerator = TRUE
   THEN
       #fault := TRUE;
       #statFault := TRUE;
       #done := FALSE;
       #busy := FALSE;
   END_IF;

   IF #reset = TRUE THEN
       #done := FALSE;
       #fault := FALSE;
       #statFault := FALSE;
       #statStageWarm := 0;
   END_IF;


   // Проверка по времени выполнения команды программирования тока и напряжения
   "IEC_Timer_0_DB_10".TON(IN := #statTimeBrakeEN,
                           PT := T#1s,
                           Q => #statTimeBrakeWarm);


   // Отсчет времени выполнения очередной стадии прогрева
   "IEC_Timer_0_DB_9".TON(IN:=#statTimeStageEn,
                          PT:=#statTime,
                          Q=>#statStageDone,
                          ET=>#statTimeOff);

   //Вычисляем остаток времени прогрева
   IF #statStageWarm > 0  THEN
       #TimeOut := #statTimeOveral - #statTime * (#statStageWarm - 1) - #statTimeOff;
   END_IF;

   IF #statStageDone = TRUE THEN
       #statStageWarm := #statStageWarm + 1;
   END_IF;
END_FUNCTION_BLOCK

FUNCTION_BLOCK "GeneratorDIO"   // FB3, SCL
{ S7_Optimized_Access := 'TRUE' }
VERSION : 0.1
   VAR_INPUT
      enable : Bool;
      reset : Bool;
      port : Port;
      debug : Bool;   // Debug Flag
   END_VAR
   VAR_OUTPUT
      done : Bool;   // TRUE: Command execuite without error
      done_CMD : UInt;
      error : Bool;   // TRUE: An error occurred during the execution of the FB
      status : Word := 16#7000;   // 16#0000 - 16#7FFF: Status of the FB, 16#8000 - 16#FFFF: Error identification
   END_VAR
   VAR_IN_OUT
      DATA : "typeGeneratorDATA";
   END_VAR
   VAR
      statCMDState : UInt := 0;   // State in the state machine of the FB
      statCMDCount : UInt := 0;   // State in the state machine of the FB
      statCMDSendReq : Bool;
      statCMDStateDone : UInt;
      statConvertData : Array[0..10] of Char;   // Convertion Data Buffer
      statString : String[30];
      statCHARtoHEX : UInt;
      statCountChar : UInt;
      statSendData : Array[0..20] of Byte;   // Sent Data
      statRcvData : Array[0..50] of Byte;   // Received Data
      statSendReq : Bool;   // Enable Send_P2P
      statSendTxLength : UInt;   // Length of Data
      statSendRxLength : UInt;   // Length of Data
      statRS232TxDone : Bool;
      statRS232Error : Bool;
      statRS232Status : Word;
      statRS232Ndr : Bool;   // Static value for output 'ndr'
      statError : Bool;   // Static value for output 'error'
      statStatus : Word;   // Static value for output 'status'
      instSendP2P : Send_P2P;   // Instance of Send_P2P
      instReceiveP2P : Receive_P2P;   // Instance of Receive_P2P
   END_VAR
   VAR_TEMP
      tempReset : Bool;
      tempEnable : Bool;
      statResetOld : Bool;
      statEnableOld : Bool;   // Old value of 'enable' input for edge detection
      temp_Uint : UInt;
   END_VAR
   VAR CONSTANT
      FB_STATE_NO_PROCESSING : UInt := 0;   // FB state: No processing
      FB_STATE_VOLTAGE_PROGRAMM : UInt := 1;   // FB state: Set Voltage / FB state: Reader RF1070R Initialization
      FB_STATE_CURRENT_PROGRAMM : UInt := 2;   // FB state: Set Current / FB state: Waiting forreset response
      FB_STATE_MONITOR : UInt := 3;   // FB state: Monitor
      FB_STATE_FAULT_CLEAR : UInt := 4;   // FB state: Fault Clear / FB state: Waiting forreset response
      FB_STATE_REPORT_FAULT : UInt := 5;   // FB state: Report Fault / FB state: Waiting forreset response
      FB_STATE_HV_STATUS : UInt := 6;   // FB state: HV Status / FB state: Waiting forreset response
      FB_STATE_X_RAY_ENABLE : UInt := 7;   // FB state: X-RAY Enable / FB state: Waiting forreset response
      FB_STATE_WD_TIMER : UInt := 8;   // FB state: Wath DOG Timer / FB state: Waiting forreset response
      FB_STATE_COMM_PORT_ECHO : UInt := 9;   // FB state: Comm Port Echo / FB state: Waiting forreset response
      FB_STATE_WD_ENABLE : UInt := 10;   // FB state: Watch Dog Enable/Disable / FB state: Waiting forreset response
      FB_STATE_WD_STATUS : UInt := 11;   // FB state: Watch Dog / FB state: Waiting forreset response
      FB_STATE_ENABLING : UInt := 12;   // FB state: Enabling
      STATUS_msg_timeout : Word := 16#0095;
      STATUS_NO_CALL : Word := 16#7000;   // No job being currently processed
      ERR_Response_Generator : Word := 16#8701;   // Error: response from generator not match argument CMD
   END_VAR
BEGIN
       REGION BLOCK INFO HEADER
       //===============================================================================
       // (company) / (c)Copyright (year)
       //-------------------------------------------------------------------------------
       // Title:            GENER
       // Comment/Function: Read out the VJ X-ray generator
       // Library/Family:   
       // Author:           Matskevich
       // Tested with:      CPU 1214C , CM1241 RS232 V2.2
       // Engineering:      TIA V15.1, update 3
       // Restrictions:     OB100, OB1
       // Requirements:     CPU 1214C , CM1241 RS232 V2.2
       //-------------------------------------------------------------------------------
       // Change log table:
       // Version  | Date       | Expert in charge       | Changes applied
       //----------|------------|------------------------|------------------------------
       // 01.00.00 | 2021-01-09 |                        | First released version
       //===============================================================================
   END_REGION
   #tempReset := #reset;   // Work with temporary value / create process image
   #tempEnable := #enable;

   REGION ENABLING/DISABLING

       IF (#tempReset = TRUE) AND (NOT #statResetOld) THEN // Reset 
           // First call; initialize FB
           #statCMDState := #FB_STATE_ENABLING;
           #statError := FALSE;
           #statRS232Ndr := FALSE;
           #statCMDCount := 0;
           #statStatus := 0;
           #statSendReq := FALSE;
           #statCMDStateDone := 0;
           #done := FALSE;
           #done_CMD := 0;
           #DATA.CMD_VP := FALSE;
           #DATA.CMD_CP := FALSE;
           #DATA.CMD_MON := FALSE;
           #DATA.CMD_CLR := FALSE;
           #DATA.CMD_FLT := FALSE;
           #DATA.CMD_STAT := FALSE;
           #DATA.CMD_ENBL := FALSE;
           #DATA.CMD_WDTE := FALSE;
           #DATA.CMD_FREV := FALSE;
           #DATA.CMD_WDOG := FALSE;
           #DATA.CMD_STAT := FALSE;
           #DATA.CMD_WSTAT := FALSE;
           #DATA.FREV := FALSE;

           FILL_BLK(IN := 16#00,
                    COUNT := 20,
                    OUT => #statSendData[0]);

           FILL_BLK(IN := 16#00,
                    COUNT := 50,
                    OUT => #statRcvData[0]);
           #instReceiveP2P.LENGTH := 0;
           #statStatus := "STATUS_RESET_END";

       ELSIF (#tempEnable = TRUE) AND (#statCMDState = #FB_STATE_NO_PROCESSING) THEN // Enable FB
           // First call; initialize FB
           ;
       ELSIF (#tempEnable = FALSE) AND (#statEnableOld = TRUE) THEN // Disable FB 
           #statCMDState := #STATUS_NO_CALL;

       END_IF;

       // Edge detection 'reset' input
       #statResetOld := #tempReset;
       // Edge detection 'enable' input
       #statEnableOld := #tempEnable;

   END_REGION ENABLING/DISABLING

   IF #statSendReq = TRUE THEN
       #statSendReq := FALSE;
   END_IF;

   IF (#statStatus = #STATUS_NO_CALL) THEN // Nothing to do -> End here to reduce "system load"
       RETURN;
   END_IF;

   REGION STATE_MACHINE

       CASE #statCMDState OF

           #FB_STATE_NO_PROCESSING:
               ;

           #FB_STATE_ENABLING: // Enabling active
               REGION enablin         
                   #statCMDState := #FB_STATE_VOLTAGE_PROGRAMM;
                   #statCMDCount := 0;
               END_REGION enabling  

           #FB_STATE_VOLTAGE_PROGRAMM:
               REGION VOLTAGE_PROGRAMM  
                   IF #DATA.CMD_VP = 1 THEN
                       IF ("CycleInterrupt_Flag" = TRUE)
                       THEN
                           #done := FALSE;
                           "CycleInterrupt_Flag" := FALSE;
                           #statCMDStateDone := #FB_STATE_VOLTAGE_PROGRAMM;
                           FILL_BLK(IN := 16#00,
                                    COUNT := 20,
                                    OUT => #statSendData[0]);

                           #statSendData[0] := 16#02;
                           #statSendData[1] := 'V';
                           #statSendData[2] := 'P';

                           //Преобразовываем из UInt в ASCII
                           // VP (Real XXX.X) -> VP*10 (Real XXXХ.X) -> temp_VP (uint XXXX) -> statSendData[3] (ASCII 4-е байта)
                           #temp_Uint := REAL_TO_UINT(#DATA.VP_Programm * 10);
                           VAL_STRG(IN := #temp_Uint,
                                    SIZE := 10,
                                    PREC := 0,
                                    FORMAT := 0,
                                    P := 1,
                                    OUT => #statString);
                           Strg_TO_Chars(Strg := #statString,
                                         pChars := 0,
                                         Cnt => #statCountChar,
                                         Chars := #statConvertData);


                           #statSendData[3] := #statConvertData[6];
                           #statSendData[4] := #statConvertData[7];
                           #statSendData[5] := #statConvertData[8];
                           #statSendData[6] := #statConvertData[9];

                           IF #statSendData[3] = ' ' THEN
                               #statSendData[3] := '0';
                           END_IF;
                           IF #statSendData[4] = ' ' THEN
                               #statSendData[4] := '0';
                           END_IF;
                           IF #statSendData[5] = ' ' THEN
                               #statSendData[5] := '0';
                           END_IF;
                           IF #statSendData[6] = ' ' THEN
                               #statSendData[6] := '0';
                           END_IF;

                           #statSendData[7] := 16#0D;
                           #statSendTxLength := 8;

                           #statSendReq := TRUE;
                       END_IF;

                   ELSE
                       #statCMDCount := 0;
                       #statCMDState := #statCMDState + 1;
                   END_IF;

               END_REGION VOLTAGE_PROGRAMM    

           #FB_STATE_CURRENT_PROGRAMM:
               REGION CURRENT_PROGRAMM
                   IF #DATA.CMD_CP = 1 THEN
                       IF ("CycleInterrupt_Flag" = TRUE)
                       THEN
                           "CycleInterrupt_Flag" := FALSE;
                           #done := FALSE;
                           #statCMDStateDone := #FB_STATE_CURRENT_PROGRAMM;
                           FILL_BLK(IN := 16#00,
                                    COUNT := 20,
                                    OUT => #statSendData[0]);

                           #statSendData[0] := 16#02;
                           #statSendData[1] := 'C';
                           #statSendData[2] := 'P';

                           //Преобразовываем из UInt в ASCII
                           // CP (Real XXX.X) -> temp_VP (uint XXXX) -> statSendData[3] (ASCII 4-е байта)
                           #temp_Uint := REAL_TO_UINT(#DATA.CP_Programm);
                           VAL_STRG(IN := #temp_Uint,
                                    SIZE := 10,
                                    PREC := 0,
                                    FORMAT := 0,
                                    P := 1,
                                    OUT => #statString);
                           Strg_TO_Chars(Strg := #statString,
                                         pChars := 0,
                                         Cnt => #statCountChar,
                                         Chars := #statConvertData);

                           #statSendData[3] := #statConvertData[6];
                           #statSendData[4] := #statConvertData[7];
                           #statSendData[5] := #statConvertData[8];
                           #statSendData[6] := #statConvertData[9];

                           IF #statSendData[3] = ' ' THEN
                               #statSendData[3] := '0';
                           END_IF;
                           IF #statSendData[4] = ' ' THEN
                               #statSendData[4] := '0';
                           END_IF;
                           IF #statSendData[5] = ' ' THEN
                               #statSendData[5] := '0';
                           END_IF;
                           IF #statSendData[6] = ' ' THEN
                               #statSendData[6] := '0';
                           END_IF;

                           #statSendData[7] := 16#0D;
                           #statSendTxLength := 8;

                           #statSendReq := TRUE;
                       END_IF;

                   ELSE
                       #statCMDCount := 0;
                       #statCMDState := #statCMDState + 1;
                   END_IF;

               END_REGION CURRENT_PROGRAMM

